KUKA KRL program: f1_Kuka_APT229T02S29.SRC

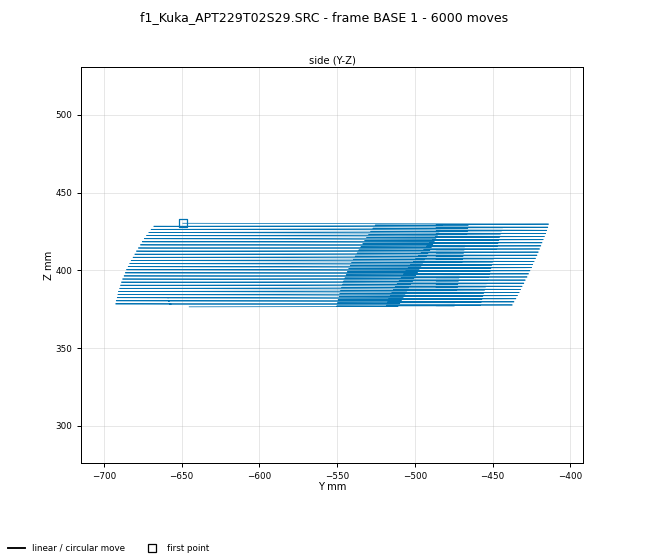
[picture p0: tool path of f1_Kuka_APT229T02S29.SRC in frame BASE 1, 6000 of 6001 moves have a stored position in this frame; points joined in program order, loops and branches not executed]
&ACCESS RVP
&REL 2
&PARAM TEMPLATE = C:\KRC\Roboter\Template\vorgabe
&PARAM EDITMASK = *
DEF f1_Kuka_APT229T02S29()


;FOLD INI;%{PE}%V3.2.0,%MKUKATPBASIS,%CINIT,%VCOMMON,%P
  ;FOLD BAS INI;%{E}%V3.2.0,%MKUKATPBASIS,%CINIT,%VINIT,%P
    GLOBAL INTERRUPT DECL 3 WHEN $STOPMESS==TRUE DO IR_STOPM ( )
    INTERRUPT ON 3
    BAS (#INITMOV,0 )
  ;ENDFOLD (BAS INI)
  ;FOLD USER INI;%{E}%V3.2.0,%MKUKATPUSER,%CINIT,%VINIT,%P
    ;Make your modifications here
  ;ENDFOLD (USER INI)
;ENDFOLD (INI)


;*** Make Null PTP Move
  PTP $pos_act

;*** Auto Load The Correct TOOL Data
  $tool=tool_data[2]

;*** Auto Load The Correct BASE Data
  $base=base_data[1]

  $ADVANCE = 5

;*** Restate Last Velocity
MMPM(30000.0)
SetRPM(8000)
LIN {X -0.016,Y -649.199,Z 430.291,A 0.000,B 0.000,C 90.000,E1 268.453} C_DIS
LIN {X 0.217,Y -646.027,Z 430.285,A 0.000,B 0.000,C 90.000,E1 267.192} C_DIS
LIN {X -0.248,Y -642.645,Z 430.278,A 0.000,B 0.000,C 90.000,E1 265.988} C_DIS
LIN {X 0.108,Y -637.908,Z 430.268,A 0.000,B 0.000,C 90.000,E1 264.204} C_DIS
LIN {X -0.169,Y -635.019,Z 430.262,A 0.000,B 0.000,C 90.000,E1 263.223} C_DIS
LIN {X -0.343,Y -630.490,Z 430.254,A 0.000,B 0.000,C 90.000,E1 261.724} C_DIS
LIN {X 0.198,Y -625.800,Z 430.245,A 0.000,B 0.000,C 90.000,E1 260.151} C_DIS
LIN {X 0.256,Y -621.879,Z 430.238,A 0.000,B 0.000,C 90.000,E1 258.870} C_DIS
LIN {X 0.011,Y -617.013,Z 430.230,A 0.000,B 0.000,C 90.000,E1 257.353} C_DIS
LIN {X 0.035,Y -612.805,Z 430.223,A 0.000,B 0.000,C 90.000,E1 256.061} C_DIS
LIN {X 0.137,Y -608.499,Z 430.215,A 0.000,B 0.000,C 90.000,E1 254.755} C_DIS
LIN {X 0.065,Y -603.102,Z 430.207,A 0.000,B 0.000,C 90.000,E1 253.196} C_DIS
LIN {X -0.110,Y -597.511,Z 430.198,A 0.000,B 0.000,C 90.000,E1 251.638} C_DIS
LIN {X -0.101,Y -592.747,Z 430.191,A 0.000,B 0.000,C 90.000,E1 250.315} C_DIS
LIN {X 0.225,Y -587.839,Z 430.183,A 0.000,B 0.000,C 90.000,E1 248.954} C_DIS
LIN {X -0.158,Y -583.761,Z 430.177,A 0.000,B 0.000,C 90.000,E1 247.922} C_DIS
LIN {X 0.241,Y -578.506,Z 430.170,A 0.000,B 0.000,C 90.000,E1 246.538} C_DIS
LIN {X -0.209,Y -573.098,Z 430.162,A 0.000,B 0.000,C 90.000,E1 245.229} C_DIS
LIN {X 0.076,Y -566.512,Z 430.153,A 0.000,B 0.000,C 90.000,E1 243.563} C_DIS
LIN {X -0.343,Y -561.046,Z 430.146,A 0.000,B 0.000,C 90.000,E1 242.231} C_DIS
LIN {X -0.009,Y -553.450,Z 430.135,A 0.000,B 0.000,C 90.000,E1 240.255} C_DIS
LIN {X 0.126,Y -546.096,Z 430.124,A 0.000,B 0.000,C 90.000,E1 238.280} C_DIS
LIN {X 0.161,Y -539.936,Z 430.114,A 0.000,B 0.000,C 90.000,E1 236.580} C_DIS
LIN {X -0.077,Y -532.802,Z 430.103,A 0.000,B 0.000,C 90.000,E1 234.609} C_DIS
LIN {X 0.300,Y -527.842,Z 430.095,A 0.000,B 0.000,C 90.000,E1 233.130} C_DIS
LIN {X 0.113,Y -521.840,Z 430.086,A 0.000,B 0.000,C 90.000,E1 231.412} C_DIS
LIN {X -0.126,Y -510.774,Z 430.066,A 0.000,B 0.000,C 90.000,E1 227.919} C_DIS
LIN {X -0.080,Y -505.592,Z 430.056,A 0.000,B 0.000,C 90.000,E1 226.134} C_DIS
LIN {X -0.164,Y -500.522,Z 430.046,A 0.000,B 0.000,C 90.000,E1 224.352} C_DIS
LIN {X 0.181,Y -494.664,Z 430.035,A 0.000,B 0.000,C 90.000,E1 222.204} C_DIS
LIN {X 0.227,Y -491.411,Z 430.028,A 0.000,B 0.000,C 90.000,E1 220.987} C_DIS
LIN {X 0.238,Y -485.107,Z 430.014,A 0.000,B 0.000,C 90.000,E1 218.543} C_DIS
LIN {X -0.168,Y -482.013,Z 430.008,A 0.000,B 0.000,C 90.000,E1 217.363} C_DIS
LIN {X -0.047,Y -478.278,Z 429.999,A 0.000,B 0.000,C 90.000,E1 215.804} C_DIS
LIN {X 0.000,Y -474.711,Z 429.990,A 0.000,B 0.000,C 90.000,E1 214.246} C_DIS
LIN {X 0.270,Y -470.560,Z 429.980,A 0.000,B 0.000,C 90.000,E1 212.339} C_DIS
LIN {X 0.198,Y -466.398,Z 429.969,A 0.000,B 0.000,C 90.000,E1 210.463} C_DIS
LIN {X 0.152,Y -463.698,Z 429.962,A 0.000,B 0.000,C 90.000,E1 209.205} C_DIS
LIN {X -0.031,Y -460.266,Z 429.954,A 0.000,B 0.000,C 90.000,E1 207.641} C_DIS
LIN {X -0.073,Y -455.343,Z 429.941,A 0.000,B 0.000,C 90.000,E1 205.412} C_DIS
LIN {X 0.200,Y -451.801,Z 429.932,A 0.000,B 0.000,C 90.000,E1 203.770} C_DIS
LIN {X 0.098,Y -447.565,Z 429.921,A 0.000,B 0.000,C 90.000,E1 201.844} C_DIS
LIN {X 0.136,Y -441.419,Z 429.905,A 0.000,B 0.000,C 90.000,E1 198.906} C_DIS
LIN {X -0.038,Y -436.063,Z 429.889,A 0.000,B 0.000,C 90.000,E1 195.969} C_DIS
LIN {X -0.014,Y -432.177,Z 429.876,A 0.000,B 0.000,C 90.000,E1 193.647} C_DIS
LIN {X -0.008,Y -427.119,Z 429.857,A 0.000,B 0.000,C 90.000,E1 190.310} C_DIS
LIN {X -0.166,Y -423.653,Z 429.842,A 0.000,B 0.000,C 90.000,E1 187.644} C_DIS
LIN {X -0.143,Y -420.857,Z 429.829,A 0.000,B 0.000,C 90.000,E1 185.277} C_DIS
LIN {X 0.063,Y -419.125,Z 429.820,A 0.000,B 0.000,C 90.000,E1 183.555} C_DIS
LIN {X -0.120,Y -416.780,Z 429.805,A 0.000,B 0.000,C 90.000,E1 180.859} C_DIS
LIN {X 0.009,Y -415.250,Z 429.791,A 0.000,B 0.000,C 90.000,E1 178.453} C_DIS
LIN {X 0.188,Y -414.001,Z 429.772,A 0.000,B 0.000,C 90.000,E1 175.008} C_DIS
LIN {X 0.130,Y -413.945,Z 429.750,A 0.000,B 0.000,C 90.000,E1 170.905} C_DIS
LIN {X 0.120,Y -414.832,Z 429.733,A 0.000,B 0.000,C 90.000,E1 167.825} C_DIS
LIN {X -0.129,Y -417.090,Z 429.712,A 0.000,B 0.000,C 90.000,E1 164.102} C_DIS
LIN {X -0.134,Y -419.840,Z 429.695,A 0.000,B 0.000,C 90.000,E1 161.040} C_DIS
LIN {X 0.203,Y -422.896,Z 429.680,A 0.000,B 0.000,C 90.000,E1 158.284} C_DIS
LIN {X 0.016,Y -426.446,Z 429.665,A 0.000,B 0.000,C 90.000,E1 155.613} C_DIS
LIN {X 0.098,Y -429.955,Z 429.652,A 0.000,B 0.000,C 90.000,E1 153.256} C_DIS
LIN {X -0.105,Y -432.179,Z 429.644,A 0.000,B 0.000,C 90.000,E1 151.948} C_DIS
LIN {X -0.048,Y -436.379,Z 429.631,A 0.000,B 0.000,C 90.000,E1 149.616} C_DIS
LIN {X 0.080,Y -441.687,Z 429.617,A 0.000,B 0.000,C 90.000,E1 146.962} C_DIS
LIN {X -0.047,Y -446.659,Z 429.604,A 0.000,B 0.000,C 90.000,E1 144.689} C_DIS
LIN {X -0.105,Y -454.457,Z 429.586,A 0.000,B 0.000,C 90.000,E1 141.457} C_DIS
LIN {X 0.086,Y -458.636,Z 429.577,A 0.000,B 0.000,C 90.000,E1 139.828} C_DIS
LIN {X 0.005,Y -462.850,Z 429.568,A 0.000,B 0.000,C 90.000,E1 138.243} C_DIS
LIN {X -0.151,Y -465.356,Z 429.563,A 0.000,B 0.000,C 90.000,E1 137.310} C_DIS
LIN {X -0.213,Y -468.530,Z 429.556,A 0.000,B 0.000,C 90.000,E1 136.053} C_DIS
LIN {X 0.190,Y -472.118,Z 429.547,A 0.000,B 0.000,C 90.000,E1 134.433} C_DIS
LIN {X -0.110,Y -474.684,Z 429.540,A 0.000,B 0.000,C 90.000,E1 133.218} C_DIS
LIN {X -0.237,Y -475.760,Z 429.537,A 0.000,B 0.000,C 90.000,E1 132.609} C_DIS
LIN {X -0.249,Y -477.194,Z 429.531,A 0.000,B 0.000,C 90.000,E1 131.676} C_DIS
LIN {X 0.115,Y -478.293,Z 429.526,A 0.000,B 0.000,C 90.000,E1 130.701} C_DIS
LIN {X -0.181,Y -478.951,Z 429.521,A 0.000,B 0.000,C 90.000,E1 129.806} C_DIS
LIN {X -0.074,Y -479.116,Z 429.519,A 0.000,B 0.000,C 90.000,E1 129.483} C_DIS
LIN {X 0.010,Y -479.158,Z 429.514,A 0.000,B 0.000,C 90.000,E1 128.543} C_DIS
LIN {X 0.097,Y -478.631,Z 429.509,A 0.000,B 0.000,C 90.000,E1 127.604} C_DIS
LIN {X 0.180,Y -477.585,Z 429.504,A 0.000,B 0.000,C 90.000,E1 126.664} C_DIS
LIN {X 0.246,Y -476.278,Z 429.499,A 0.000,B 0.000,C 90.000,E1 125.724} C_DIS
LIN {X 0.224,Y -475.231,Z 429.495,A 0.000,B 0.000,C 90.000,E1 125.105} C_DIS
LIN {X -0.193,Y -473.865,Z 429.492,A 0.000,B 0.000,C 90.000,E1 124.532} C_DIS
LIN {X -0.054,Y -471.563,Z 429.487,A 0.000,B 0.000,C 90.000,E1 123.579} C_DIS
LIN {X 0.061,Y -468.905,Z 429.481,A 0.000,B 0.000,C 90.000,E1 122.625} C_DIS
LIN {X -0.103,Y -464.908,Z 429.474,A 0.000,B 0.000,C 90.000,E1 121.386} C_DIS
LIN {X 0.090,Y -461.619,Z 429.469,A 0.000,B 0.000,C 90.000,E1 120.413} C_DIS
LIN {X -0.027,Y -456.831,Z 429.462,A 0.000,B 0.000,C 90.000,E1 119.155} C_DIS
LIN {X -0.090,Y -451.157,Z 429.454,A 0.000,B 0.000,C 90.000,E1 117.719} C_DIS
LIN {X 0.140,Y -445.297,Z 429.446,A 0.000,B 0.000,C 90.000,E1 116.232} C_DIS
LIN {X 0.209,Y -442.718,Z 429.442,A 0.000,B 0.000,C 90.000,E1 115.591} C_DIS
LIN {X 0.169,Y -442.732,Z 429.442,A 0.000,B 0.000,C 90.000,E1 115.591} C_DIS
LIN {X -0.059,Y -444.742,Z 429.439,A 0.000,B 0.000,C 90.000,E1 114.951} C_DIS
LIN {X -0.088,Y -454.712,Z 429.415,A 0.000,B 0.000,C 90.000,E1 110.737} C_DIS
LIN {X 0.035,Y -457.355,Z 429.410,A 0.000,B 0.000,C 90.000,E1 109.758} C_DIS
LIN {X 0.120,Y -465.984,Z 429.387,A 0.000,B 0.000,C 90.000,E1 105.607} C_DIS
LIN {X -0.158,Y -467.550,Z 429.383,A 0.000,B 0.000,C 90.000,E1 105.009} C_DIS
LIN {X 0.026,Y -468.567,Z 429.380,A 0.000,B 0.000,C 90.000,E1 104.356} C_DIS
LIN {X -0.215,Y -475.787,Z 429.357,A 0.000,B 0.000,C 90.000,E1 100.310} C_DIS
LIN {X 0.091,Y -476.298,Z 429.355,A 0.000,B 0.000,C 90.000,E1 99.962} C_DIS
LIN {X 0.039,Y -481.778,Z 429.331,A 0.000,B 0.000,C 90.000,E1 95.625} C_DIS
LIN {X -0.114,Y -482.169,Z 429.330,A 0.000,B 0.000,C 90.000,E1 95.334} C_DIS
LIN {X -0.185,Y -485.300,Z 429.306,A 0.000,B 0.000,C 90.000,E1 91.031} C_DIS
LIN {X 0.125,Y -485.537,Z 429.304,A 0.000,B 0.000,C 90.000,E1 90.688} C_DIS
LIN {X -0.153,Y -486.316,Z 429.282,A 0.000,B 0.000,C 90.000,E1 86.731} C_DIS
LIN {X -0.018,Y -486.309,Z 429.278,A 0.000,B 0.000,C 90.000,E1 86.102} C_DIS
LIN {X 0.186,Y -484.696,Z 429.255,A 0.000,B 0.000,C 90.000,E1 81.781} C_DIS
LIN {X 0.055,Y -484.608,Z 429.253,A 0.000,B 0.000,C 90.000,E1 81.489} C_DIS
LIN {X -0.065,Y -480.540,Z 429.227,A 0.000,B 0.000,C 90.000,E1 76.881} C_DIS
LIN {X -0.154,Y -474.292,Z 429.201,A 0.000,B 0.000,C 90.000,E1 72.236} C_DIS
LIN {X 0.117,Y -473.862,Z 429.200,A 0.000,B 0.000,C 90.000,E1 71.891} C_DIS
LIN {X -0.206,Y -466.265,Z 429.175,A 0.000,B 0.000,C 90.000,E1 67.539} C_DIS
LIN {X -0.277,Y -465.558,Z 429.172,A 0.000,B 0.000,C 90.000,E1 67.050} C_DIS
LIN {X 0.111,Y -465.576,Z 429.172,A 0.000,B 0.000,C 90.000,E1 66.997} C_DIS
LIN {X -0.066,Y -477.055,Z 429.164,A 0.000,B 0.000,C 90.000,E1 65.485} C_DIS
LIN {X -0.139,Y -485.128,Z 429.158,A 0.000,B 0.000,C 90.000,E1 64.409} C_DIS
LIN {X 0.101,Y -491.924,Z 429.153,A 0.000,B 0.000,C 90.000,E1 63.461} C_DIS
LIN {X -0.263,Y -497.100,Z 429.148,A 0.000,B 0.000,C 90.000,E1 62.743} C_DIS
LIN {X 0.056,Y -500.940,Z 429.145,A 0.000,B 0.000,C 90.000,E1 62.103} C_DIS
LIN {X -0.038,Y -504.550,Z 429.142,A 0.000,B 0.000,C 90.000,E1 61.513} C_DIS
LIN {X -0.104,Y -507.850,Z 429.138,A 0.000,B 0.000,C 90.000,E1 60.923} C_DIS
LIN {X -0.146,Y -510.859,Z 429.135,A 0.000,B 0.000,C 90.000,E1 60.333} C_DIS
LIN {X 0.010,Y -513.067,Z 429.133,A 0.000,B 0.000,C 90.000,E1 59.871} C_DIS
LIN {X 0.004,Y -515.608,Z 429.129,A 0.000,B 0.000,C 90.000,E1 59.282} C_DIS
LIN {X 0.281,Y -517.787,Z 429.126,A 0.000,B 0.000,C 90.000,E1 58.663} C_DIS
LIN {X -0.065,Y -518.781,Z 429.124,A 0.000,B 0.000,C 90.000,E1 58.408} C_DIS
LIN {X 0.238,Y -520.483,Z 429.121,A 0.000,B 0.000,C 90.000,E1 57.788} C_DIS
LIN {X 0.223,Y -522.504,Z 429.116,A 0.000,B 0.000,C 90.000,E1 56.914} C_DIS
LIN {X 0.124,Y -523.546,Z 429.113,A 0.000,B 0.000,C 90.000,E1 56.342} C_DIS
LIN {X 0.136,Y -524.629,Z 429.108,A 0.000,B 0.000,C 90.000,E1 55.468} C_DIS
LIN {X 0.023,Y -525.268,Z 429.103,A 0.000,B 0.000,C 90.000,E1 54.609} C_DIS
LIN {X -0.076,Y -525.472,Z 429.099,A 0.000,B 0.000,C 90.000,E1 53.749} C_DIS
LIN {X 0.248,Y -525.326,Z 429.094,A 0.000,B 0.000,C 90.000,E1 52.844} C_DIS
LIN {X 0.145,Y -524.993,Z 429.089,A 0.000,B 0.000,C 90.000,E1 51.984} C_DIS
LIN {X 0.326,Y -524.156,Z 429.082,A 0.000,B 0.000,C 90.000,E1 50.803} C_DIS
LIN {X 0.094,Y -523.105,Z 429.076,A 0.000,B 0.000,C 90.000,E1 49.666} C_DIS
LIN {X -0.149,Y -521.838,Z 429.070,A 0.000,B 0.000,C 90.000,E1 48.528} C_DIS
LIN {X 0.322,Y -520.387,Z 429.063,A 0.000,B 0.000,C 90.000,E1 47.310} C_DIS
LIN {X 0.219,Y -518.084,Z 429.053,A 0.000,B 0.000,C 90.000,E1 45.567} C_DIS
LIN {X -0.032,Y -515.626,Z 429.042,A 0.000,B 0.000,C 90.000,E1 43.542} C_DIS
LIN {X 0.137,Y -513.685,Z 429.032,A 0.000,B 0.000,C 90.000,E1 41.757} C_DIS
LIN {X -0.162,Y -511.433,Z 429.021,A 0.000,B 0.000,C 90.000,E1 39.725} C_DIS
LIN {X 0.050,Y -509.857,Z 429.012,A 0.000,B 0.000,C 90.000,E1 38.222} C_DIS
LIN {X -0.088,Y -507.810,Z 429.003,A 0.000,B 0.000,C 90.000,E1 36.457} C_DIS
LIN {X 0.132,Y -506.032,Z 428.994,A 0.000,B 0.000,C 90.000,E1 34.945} C_DIS
LIN {X -0.156,Y -504.549,Z 428.988,A 0.000,B 0.000,C 90.000,E1 33.785} C_DIS
LIN {X -0.272,Y -502.186,Z 428.978,A 0.000,B 0.000,C 90.000,E1 32.005} C_DIS
LIN {X -0.281,Y -499.794,Z 428.968,A 0.000,B 0.000,C 90.000,E1 30.207} C_DIS
LIN {X 0.199,Y -498.176,Z 428.961,A 0.000,B 0.000,C 90.000,E1 28.949} C_DIS
LIN {X -0.153,Y -495.846,Z 428.951,A 0.000,B 0.000,C 90.000,E1 27.180} C_DIS
LIN {X 0.137,Y -493.409,Z 428.939,A 0.000,B 0.000,C 90.000,E1 25.027} C_DIS
LIN {X -0.177,Y -490.454,Z 428.922,A 0.000,B 0.000,C 90.000,E1 22.025} C_DIS
LIN {X -0.133,Y -488.913,Z 428.910,A 0.000,B 0.000,C 90.000,E1 19.885} C_DIS
LIN {X -0.155,Y -487.703,Z 428.900,A 0.000,B 0.000,C 90.000,E1 18.055} C_DIS
LIN {X 0.085,Y -486.635,Z 428.892,A 0.000,B 0.000,C 90.000,E1 16.496} C_DIS
LIN {X 0.036,Y -485.106,Z 428.880,A 0.000,B 0.000,C 90.000,E1 14.356} C_DIS
LIN {X 0.027,Y -483.620,Z 428.864,A 0.000,B 0.000,C 90.000,E1 11.591} C_DIS
LIN {X -0.164,Y -483.028,Z 428.856,A 0.000,B 0.000,C 90.000,E1 10.074} C_DIS
LIN {X 0.025,Y -482.452,Z 428.842,A 0.000,B 0.000,C 90.000,E1 7.587} C_DIS
LIN {X -0.200,Y -482.436,Z 428.825,A 0.000,B 0.000,C 90.000,E1 4.531} C_DIS
LIN {X -0.119,Y -483.946,Z 428.803,A 0.000,B 0.000,C 90.000,E1 0.516} C_DIS
LIN {X 0.070,Y -488.037,Z 428.778,A 0.000,B 0.000,C 90.000,E1 356.102} C_DIS
LIN {X -0.152,Y -491.259,Z 428.765,A 0.000,B 0.000,C 90.000,E1 353.685} C_DIS
LIN {X -0.054,Y -494.482,Z 428.753,A 0.000,B 0.000,C 90.000,E1 351.546} C_DIS
LIN {X 0.208,Y -498.075,Z 428.741,A 0.000,B 0.000,C 90.000,E1 349.398} C_DIS
LIN {X -0.115,Y -507.281,Z 428.716,A 0.000,B 0.000,C 90.000,E1 344.936} C_DIS
LIN {X -0.011,Y -511.555,Z 428.706,A 0.000,B 0.000,C 90.000,E1 343.142} C_DIS
LIN {X -0.046,Y -517.550,Z 428.693,A 0.000,B 0.000,C 90.000,E1 340.786} C_DIS
LIN {X -0.153,Y -520.743,Z 428.687,A 0.000,B 0.000,C 90.000,E1 339.625} C_DIS
LIN {X 0.277,Y -526.392,Z 428.675,A 0.000,B 0.000,C 90.000,E1 337.539} C_DIS
LIN {X -0.110,Y -531.281,Z 428.666,A 0.000,B 0.000,C 90.000,E1 335.845} C_DIS
LIN {X 0.243,Y -537.947,Z 428.653,A 0.000,B 0.000,C 90.000,E1 333.512} C_DIS
LIN {X -0.164,Y -543.002,Z 428.644,A 0.000,B 0.000,C 90.000,E1 331.847} C_DIS
LIN {X 0.052,Y -548.210,Z 428.634,A 0.000,B 0.000,C 90.000,E1 330.127} C_DIS
LIN {X -0.132,Y -552.587,Z 428.626,A 0.000,B 0.000,C 90.000,E1 328.742} C_DIS
LIN {X 0.112,Y -557.674,Z 428.617,A 0.000,B 0.000,C 90.000,E1 327.041} C_DIS
LIN {X 0.102,Y -563.555,Z 428.606,A 0.000,B 0.000,C 90.000,E1 325.102} C_DIS
LIN {X -0.017,Y -568.641,Z 428.597,A 0.000,B 0.000,C 90.000,E1 323.463} C_DIS
LIN {X -0.030,Y -573.779,Z 428.588,A 0.000,B 0.000,C 90.000,E1 321.823} C_DIS
LIN {X -0.035,Y -579.108,Z 428.579,A 0.000,B 0.000,C 90.000,E1 320.194} C_DIS
LIN {X -0.105,Y -583.629,Z 428.571,A 0.000,B 0.000,C 90.000,E1 318.852} C_DIS
LIN {X 0.035,Y -588.923,Z 428.562,A 0.000,B 0.000,C 90.000,E1 317.229} C_DIS
LIN {X 0.087,Y -593.419,Z 428.555,A 0.000,B 0.000,C 90.000,E1 315.891} C_DIS
LIN {X -0.211,Y -597.918,Z 428.548,A 0.000,B 0.000,C 90.000,E1 314.595} C_DIS
LIN {X -0.003,Y -604.205,Z 428.537,A 0.000,B 0.000,C 90.000,E1 312.732} C_DIS
LIN {X -0.102,Y -608.674,Z 428.530,A 0.000,B 0.000,C 90.000,E1 311.434} C_DIS
LIN {X 0.344,Y -613.019,Z 428.523,A 0.000,B 0.000,C 90.000,E1 310.092} C_DIS
LIN {X 0.005,Y -617.270,Z 428.516,A 0.000,B 0.000,C 90.000,E1 308.830} C_DIS
LIN {X 0.051,Y -622.202,Z 428.507,A 0.000,B 0.000,C 90.000,E1 307.282} C_DIS
LIN {X 0.134,Y -625.268,Z 428.502,A 0.000,B 0.000,C 90.000,E1 306.251} C_DIS
LIN {X -0.048,Y -629.805,Z 428.493,A 0.000,B 0.000,C 90.000,E1 304.739} C_DIS
LIN {X 0.166,Y -633.388,Z 428.486,A 0.000,B 0.000,C 90.000,E1 303.452} C_DIS
LIN {X -0.083,Y -636.910,Z 428.479,A 0.000,B 0.000,C 90.000,E1 302.212} C_DIS
LIN {X 0.256,Y -640.311,Z 428.472,A 0.000,B 0.000,C 90.000,E1 300.924} C_DIS
LIN {X -0.171,Y -644.131,Z 428.464,A 0.000,B 0.000,C 90.000,E1 299.461} C_DIS
LIN {X -0.358,Y -647.179,Z 428.457,A 0.000,B 0.000,C 90.000,E1 298.231} C_DIS
LIN {X 0.183,Y -650.635,Z 428.448,A 0.000,B 0.000,C 90.000,E1 296.693} C_DIS
LIN {X 0.102,Y -653.383,Z 428.442,A 0.000,B 0.000,C 90.000,E1 295.463} C_DIS
LIN {X -0.228,Y -655.906,Z 428.435,A 0.000,B 0.000,C 90.000,E1 294.259} C_DIS
LIN {X -0.181,Y -658.221,Z 428.428,A 0.000,B 0.000,C 90.000,E1 293.025} C_DIS
LIN {X 0.161,Y -660.404,Z 428.421,A 0.000,B 0.000,C 90.000,E1 291.770} C_DIS
LIN {X 0.161,Y -662.106,Z 428.416,A 0.000,B 0.000,C 90.000,E1 290.791} C_DIS
LIN {X 0.185,Y -663.600,Z 428.410,A 0.000,B 0.000,C 90.000,E1 289.812} C_DIS
LIN {X 0.126,Y -665.027,Z 428.403,A 0.000,B 0.000,C 90.000,E1 288.598} C_DIS
LIN {X -0.004,Y -666.380,Z 428.395,A 0.000,B 0.000,C 90.000,E1 287.149} C_DIS
LIN {X -0.334,Y -666.984,Z 428.390,A 0.000,B 0.000,C 90.000,E1 286.205} C_DIS
LIN {X 0.176,Y -667.471,Z 428.385,A 0.000,B 0.000,C 90.000,E1 285.190} C_DIS
LIN {X -0.201,Y -667.826,Z 428.378,A 0.000,B 0.000,C 90.000,E1 284.008} C_DIS
LIN {X 0.077,Y -667.853,Z 428.371,A 0.000,B 0.000,C 90.000,E1 282.771} C_DIS
LIN {X -0.227,Y -667.796,Z 428.366,A 0.000,B 0.000,C 90.000,E1 281.827} C_DIS
LIN {X -0.017,Y -667.526,Z 428.360,A 0.000,B 0.000,C 90.000,E1 280.838} C_DIS
LIN {X 0.195,Y -667.169,Z 428.355,A 0.000,B 0.000,C 90.000,E1 279.849} C_DIS
LIN {X -0.258,Y -666.520,Z 428.349,A 0.000,B 0.000,C 90.000,E1 278.916} C_DIS
LIN {X 0.302,Y -665.478,Z 428.341,A 0.000,B 0.000,C 90.000,E1 277.409} C_DIS
LIN {X -0.277,Y -664.604,Z 428.336,A 0.000,B 0.000,C 90.000,E1 276.486} C_DIS
LIN {X 0.087,Y -662.846,Z 428.328,A 0.000,B 0.000,C 90.000,E1 274.992} C_DIS
LIN {X 0.127,Y -661.526,Z 428.322,A 0.000,B 0.000,C 90.000,E1 274.012} C_DIS
LIN {X -0.236,Y -660.847,Z 428.320,A 0.000,B 0.000,C 90.000,E1 273.555} C_DIS
LIN {X -0.166,Y -657.885,Z 428.310,A 0.000,B 0.000,C 90.000,E1 271.835} C_DIS
LIN {X 0.221,Y -655.564,Z 428.303,A 0.000,B 0.000,C 90.000,E1 270.573} C_DIS
LIN {X -0.102,Y -652.947,Z 428.297,A 0.000,B 0.000,C 90.000,E1 269.370} C_DIS
LIN {X -0.264,Y -650.618,Z 428.291,A 0.000,B 0.000,C 90.000,E1 268.396} C_DIS
LIN {X -0.006,Y -647.462,Z 428.284,A 0.000,B 0.000,C 90.000,E1 267.135} C_DIS
LIN {X 0.007,Y -643.381,Z 428.276,A 0.000,B 0.000,C 90.000,E1 265.641} C_DIS
LIN {X 0.192,Y -640.075,Z 428.269,A 0.000,B 0.000,C 90.000,E1 264.375} C_DIS
LIN {X -0.317,Y -636.524,Z 428.262,A 0.000,B 0.000,C 90.000,E1 263.166} C_DIS
LIN {X 0.254,Y -631.946,Z 428.254,A 0.000,B 0.000,C 90.000,E1 261.602} C_DIS
LIN {X -0.309,Y -628.021,Z 428.246,A 0.000,B 0.000,C 90.000,E1 260.387} C_DIS
LIN {X -0.215,Y -624.113,Z 428.239,A 0.000,B 0.000,C 90.000,E1 259.106} C_DIS
LIN {X 0.323,Y -619.233,Z 428.231,A 0.000,B 0.000,C 90.000,E1 257.521} C_DIS
LIN {X 0.027,Y -615.929,Z 428.225,A 0.000,B 0.000,C 90.000,E1 256.520} C_DIS
LIN {X -0.208,Y -610.780,Z 428.217,A 0.000,B 0.000,C 90.000,E1 254.991} C_DIS
LIN {X 0.352,Y -605.388,Z 428.208,A 0.000,B 0.000,C 90.000,E1 253.378} C_DIS
LIN {X -0.253,Y -600.766,Z 428.201,A 0.000,B 0.000,C 90.000,E1 252.127} C_DIS
LIN {X 0.006,Y -596.023,Z 428.193,A 0.000,B 0.000,C 90.000,E1 250.786} C_DIS
LIN {X 0.189,Y -591.135,Z 428.186,A 0.000,B 0.000,C 90.000,E1 249.444} C_DIS
LIN {X -0.265,Y -586.084,Z 428.179,A 0.000,B 0.000,C 90.000,E1 248.156} C_DIS
LIN {X -0.046,Y -580.839,Z 428.171,A 0.000,B 0.000,C 90.000,E1 246.794} C_DIS
LIN {X 0.067,Y -575.416,Z 428.164,A 0.000,B 0.000,C 90.000,E1 245.433} C_DIS
LIN {X -0.122,Y -568.821,Z 428.155,A 0.000,B 0.000,C 90.000,E1 243.819} C_DIS
LIN {X 0.262,Y -563.346,Z 428.147,A 0.000,B 0.000,C 90.000,E1 242.410} C_DIS
LIN {X 0.165,Y -554.657,Z 428.135,A 0.000,B 0.000,C 90.000,E1 240.205} C_DIS
LIN {X 0.140,Y -547.264,Z 428.124,A 0.000,B 0.000,C 90.000,E1 238.250} C_DIS
LIN {X -0.084,Y -541.117,Z 428.114,A 0.000,B 0.000,C 90.000,E1 236.580} C_DIS
LIN {X 0.144,Y -533.045,Z 428.102,A 0.000,B 0.000,C 90.000,E1 234.276} C_DIS
LIN {X 0.095,Y -528.088,Z 428.094,A 0.000,B 0.000,C 90.000,E1 232.844} C_DIS
LIN {X -0.045,Y -523.100,Z 428.086,A 0.000,B 0.000,C 90.000,E1 231.412} C_DIS
LIN {X 0.152,Y -511.992,Z 428.066,A 0.000,B 0.000,C 90.000,E1 227.877} C_DIS
LIN {X 0.081,Y -505.962,Z 428.055,A 0.000,B 0.000,C 90.000,E1 225.810} C_DIS
LIN {X 0.215,Y -500.042,Z 428.043,A 0.000,B 0.000,C 90.000,E1 223.704} C_DIS
LIN {X 0.204,Y -494.262,Z 428.031,A 0.000,B 0.000,C 90.000,E1 221.595} C_DIS
LIN {X -0.078,Y -487.834,Z 428.018,A 0.000,B 0.000,C 90.000,E1 219.197} C_DIS
LIN {X 0.064,Y -483.985,Z 428.009,A 0.000,B 0.000,C 90.000,E1 217.649} C_DIS
LIN {X 0.031,Y -479.463,Z 427.999,A 0.000,B 0.000,C 90.000,E1 215.804} C_DIS
LIN {X 0.287,Y -475.161,Z 427.989,A 0.000,B 0.000,C 90.000,E1 213.913} C_DIS
LIN {X -0.254,Y -471.705,Z 427.980,A 0.000,B 0.000,C 90.000,E1 212.418} C_DIS
LIN {X -0.133,Y -466.844,Z 427.968,A 0.000,B 0.000,C 90.000,E1 210.207} C_DIS
LIN {X -0.026,Y -463.423,Z 427.959,A 0.000,B 0.000,C 90.000,E1 208.615} C_DIS
LIN {X 0.070,Y -460.642,Z 427.952,A 0.000,B 0.000,C 90.000,E1 207.334} C_DIS
LIN {X 0.141,Y -456.396,Z 427.941,A 0.000,B 0.000,C 90.000,E1 205.412} C_DIS
LIN {X 0.019,Y -452.833,Z 427.932,A 0.000,B 0.000,C 90.000,E1 203.823} C_DIS
LIN {X 0.053,Y -449.257,Z 427.923,A 0.000,B 0.000,C 90.000,E1 202.206} C_DIS
LIN {X 0.005,Y -444.334,Z 427.911,A 0.000,B 0.000,C 90.000,E1 199.939} C_DIS
LIN {X -0.102,Y -438.086,Z 427.893,A 0.000,B 0.000,C 90.000,E1 196.677} C_DIS
LIN {X 0.166,Y -434.680,Z 427.882,A 0.000,B 0.000,C 90.000,E1 194.662} C_DIS
LIN {X 0.040,Y -430.907,Z 427.869,A 0.000,B 0.000,C 90.000,E1 192.355} C_DIS
LIN {X -0.064,Y -427.941,Z 427.858,A 0.000,B 0.000,C 90.000,E1 190.366} C_DIS
LIN {X 0.131,Y -424.855,Z 427.845,A 0.000,B 0.000,C 90.000,E1 187.992} C_DIS
LIN {X -0.157,Y -421.648,Z 427.830,A 0.000,B 0.000,C 90.000,E1 185.334} C_DIS
LIN {X 0.203,Y -418.647,Z 427.813,A 0.000,B 0.000,C 90.000,E1 182.236} C_DIS
LIN {X 0.036,Y -416.202,Z 427.794,A 0.000,B 0.000,C 90.000,E1 178.854} C_DIS
LIN {X -0.150,Y -414.691,Z 427.773,A 0.000,B 0.000,C 90.000,E1 175.122} C_DIS
LIN {X 0.058,Y -414.429,Z 427.758,A 0.000,B 0.000,C 90.000,E1 172.356} C_DIS
LIN {X 0.177,Y -414.624,Z 427.750,A 0.000,B 0.000,C 90.000,E1 170.971} C_DIS
LIN {X -0.144,Y -415.494,Z 427.733,A 0.000,B 0.000,C 90.000,E1 167.937} C_DIS
LIN {X 0.049,Y -417.772,Z 427.712,A 0.000,B 0.000,C 90.000,E1 164.157} C_DIS
LIN {X 0.076,Y -420.517,Z 427.695,A 0.000,B 0.000,C 90.000,E1 161.094} C_DIS
LIN {X 0.073,Y -423.969,Z 427.678,A 0.000,B 0.000,C 90.000,E1 158.050} C_DIS
LIN {X -0.103,Y -427.098,Z 427.665,A 0.000,B 0.000,C 90.000,E1 155.717} C_DIS
LIN {X -0.181,Y -430.654,Z 427.652,A 0.000,B 0.000,C 90.000,E1 153.384} C_DIS
LIN {X -0.127,Y -435.864,Z 427.635,A 0.000,B 0.000,C 90.000,E1 150.383} C_DIS
LIN {X 0.180,Y -441.780,Z 427.619,A 0.000,B 0.000,C 90.000,E1 147.375} C_DIS
LIN {X 0.058,Y -445.280,Z 427.610,A 0.000,B 0.000,C 90.000,E1 145.754} C_DIS
LIN {X -0.159,Y -449.760,Z 427.599,A 0.000,B 0.000,C 90.000,E1 143.829} C_DIS
LIN {X 0.178,Y -457.120,Z 427.583,A 0.000,B 0.000,C 90.000,E1 140.884} C_DIS
LIN {X 0.070,Y -461.412,Z 427.574,A 0.000,B 0.000,C 90.000,E1 139.299} C_DIS
LIN {X 0.041,Y -465.716,Z 427.565,A 0.000,B 0.000,C 90.000,E1 137.715} C_DIS
LIN {X 0.059,Y -469.788,Z 427.556,A 0.000,B 0.000,C 90.000,E1 136.134} C_DIS
LIN {X 0.061,Y -472.783,Z 427.549,A 0.000,B 0.000,C 90.000,E1 134.879} C_DIS
LIN {X 0.011,Y -474.819,Z 427.544,A 0.000,B 0.000,C 90.000,E1 133.947} C_DIS
LIN {X -0.011,Y -476.752,Z 427.539,A 0.000,B 0.000,C 90.000,E1 133.014} C_DIS
LIN {X 0.103,Y -478.776,Z 427.532,A 0.000,B 0.000,C 90.000,E1 131.757} C_DIS
LIN {X 0.011,Y -479.592,Z 427.529,A 0.000,B 0.000,C 90.000,E1 131.148} C_DIS
LIN {X -0.075,Y -480.298,Z 427.525,A 0.000,B 0.000,C 90.000,E1 130.539} C_DIS
LIN {X 0.020,Y -480.916,Z 427.520,A 0.000,B 0.000,C 90.000,E1 129.600} C_DIS
LIN {X 0.135,Y -481.095,Z 427.518,A 0.000,B 0.000,C 90.000,E1 129.277} C_DIS
LIN {X -0.133,Y -481.050,Z 427.513,A 0.000,B 0.000,C 90.000,E1 128.382} C_DIS
LIN {X -0.026,Y -480.436,Z 427.508,A 0.000,B 0.000,C 90.000,E1 127.443} C_DIS
LIN {X 0.074,Y -479.335,Z 427.503,A 0.000,B 0.000,C 90.000,E1 126.503} C_DIS
LIN {X -0.122,Y -478.003,Z 427.498,A 0.000,B 0.000,C 90.000,E1 125.598} C_DIS
LIN {X 0.146,Y -476.938,Z 427.494,A 0.000,B 0.000,C 90.000,E1 124.945} C_DIS
LIN {X -0.076,Y -474.750,Z 427.489,A 0.000,B 0.000,C 90.000,E1 124.040} C_DIS
LIN {X -0.107,Y -473.181,Z 427.486,A 0.000,B 0.000,C 90.000,E1 123.420} C_DIS
LIN {X 0.022,Y -470.439,Z 427.480,A 0.000,B 0.000,C 90.000,E1 122.467} C_DIS
LIN {X -0.128,Y -467.404,Z 427.475,A 0.000,B 0.000,C 90.000,E1 121.544} C_DIS
LIN {X -0.064,Y -464.182,Z 427.470,A 0.000,B 0.000,C 90.000,E1 120.590} C_DIS
LIN {X 0.102,Y -459.982,Z 427.464,A 0.000,B 0.000,C 90.000,E1 119.461} C_DIS
LIN {X 0.084,Y -454.305,Z 427.456,A 0.000,B 0.000,C 90.000,E1 118.025} C_DIS
LIN {X -0.115,Y -449.738,Z 427.450,A 0.000,B 0.000,C 90.000,E1 116.924} C_DIS
LIN {X -0.114,Y -443.700,Z 427.441,A 0.000,B 0.000,C 90.000,E1 115.463} C_DIS
LIN {X -0.227,Y -443.420,Z 427.441,A 0.000,B 0.000,C 90.000,E1 115.412} C_DIS
LIN {X -0.076,Y -443.434,Z 427.441,A 0.000,B 0.000,C 90.000,E1 115.387} C_DIS
LIN {X 0.189,Y -445.077,Z 427.438,A 0.000,B 0.000,C 90.000,E1 114.771} C_DIS
LIN {X -0.127,Y -454.237,Z 427.416,A 0.000,B 0.000,C 90.000,E1 110.918} C_DIS
LIN {X -0.011,Y -456.901,Z 427.411,A 0.000,B 0.000,C 90.000,E1 109.939} C_DIS
LIN {X -0.109,Y -457.615,Z 427.409,A 0.000,B 0.000,C 90.000,E1 109.631} C_DIS
LIN {X -0.023,Y -466.333,Z 427.386,A 0.000,B 0.000,C 90.000,E1 105.481} C_DIS
LIN {X 0.151,Y -467.870,Z 427.383,A 0.000,B 0.000,C 90.000,E1 104.828} C_DIS
LIN {X 0.179,Y -475.431,Z 427.358,A 0.000,B 0.000,C 90.000,E1 100.433} C_DIS
LIN {X 0.018,Y -476.081,Z 427.356,A 0.000,B 0.000,C 90.000,E1 100.141} C_DIS
LIN {X -0.179,Y -482.004,Z 427.331,A 0.000,B 0.000,C 90.000,E1 95.511} C_DIS
LIN {X -0.198,Y -482.514,Z 427.325,A 0.000,B 0.000,C 90.000,E1 94.588} C_DIS
LIN {X 0.092,Y -485.449,Z 427.305,A 0.000,B 0.000,C 90.000,E1 90.859} C_DIS
LIN {X 0.229,Y -485.505,Z 427.301,A 0.000,B 0.000,C 90.000,E1 90.229} C_DIS
LIN {X 0.125,Y -486.381,Z 427.281,A 0.000,B 0.000,C 90.000,E1 86.560} C_DIS
LIN {X -0.051,Y -486.365,Z 427.279,A 0.000,B 0.000,C 90.000,E1 86.274} C_DIS
LIN {X 0.038,Y -484.690,Z 427.254,A 0.000,B 0.000,C 90.000,E1 81.659} C_DIS
LIN {X 0.184,Y -484.073,Z 427.250,A 0.000,B 0.000,C 90.000,E1 81.027} C_DIS
LIN {X -0.161,Y -480.640,Z 427.228,A 0.000,B 0.000,C 90.000,E1 77.061} C_DIS
LIN {X -0.194,Y -480.346,Z 427.226,A 0.000,B 0.000,C 90.000,E1 76.756} C_DIS
LIN {X 0.177,Y -474.152,Z 427.200,A 0.000,B 0.000,C 90.000,E1 72.054} C_DIS
LIN {X 0.098,Y -465.895,Z 427.174,A 0.000,B 0.000,C 90.000,E1 67.230} C_DIS
LIN {X 0.058,Y -465.932,Z 427.174,A 0.000,B 0.000,C 90.000,E1 67.230} C_DIS
LIN {X 0.050,Y -479.069,Z 427.164,A 0.000,B 0.000,C 90.000,E1 65.485} C_DIS
LIN {X -0.210,Y -488.244,Z 427.157,A 0.000,B 0.000,C 90.000,E1 64.280} C_DIS
LIN {X -0.168,Y -493.847,Z 427.153,A 0.000,B 0.000,C 90.000,E1 63.512} C_DIS
LIN {X 0.127,Y -498.008,Z 427.149,A 0.000,B 0.000,C 90.000,E1 62.871} C_DIS
LIN {X 0.013,Y -501.879,Z 427.146,A 0.000,B 0.000,C 90.000,E1 62.281} C_DIS
LIN {X -0.071,Y -505.482,Z 427.143,A 0.000,B 0.000,C 90.000,E1 61.691} C_DIS
LIN {X -0.128,Y -508.812,Z 427.139,A 0.000,B 0.000,C 90.000,E1 61.101} C_DIS
LIN {X 0.284,Y -511.884,Z 427.136,A 0.000,B 0.000,C 90.000,E1 60.461} C_DIS
LIN {X -0.171,Y -514.738,Z 427.133,A 0.000,B 0.000,C 90.000,E1 59.921} C_DIS
LIN {X 0.108,Y -517.808,Z 427.129,A 0.000,B 0.000,C 90.000,E1 59.154} C_DIS
LIN {X -0.044,Y -519.912,Z 427.125,A 0.000,B 0.000,C 90.000,E1 58.584} C_DIS
LIN {X -0.004,Y -521.638,Z 427.122,A 0.000,B 0.000,C 90.000,E1 57.995} C_DIS
LIN {X -0.008,Y -523.742,Z 427.117,A 0.000,B 0.000,C 90.000,E1 57.120} C_DIS
LIN {X -0.099,Y -524.805,Z 427.114,A 0.000,B 0.000,C 90.000,E1 56.548} C_DIS
LIN {X -0.073,Y -525.937,Z 427.109,A 0.000,B 0.000,C 90.000,E1 55.674} C_DIS
LIN {X -0.172,Y -526.678,Z 427.104,A 0.000,B 0.000,C 90.000,E1 54.815} C_DIS
LIN {X 0.169,Y -526.900,Z 427.100,A 0.000,B 0.000,C 90.000,E1 53.909} C_DIS
LIN {X 0.086,Y -526.754,Z 427.095,A 0.000,B 0.000,C 90.000,E1 53.050} C_DIS
LIN {X 0.002,Y -526.426,Z 427.090,A 0.000,B 0.000,C 90.000,E1 52.190} C_DIS
LIN {X 0.206,Y -525.611,Z 427.084,A 0.000,B 0.000,C 90.000,E1 51.009} C_DIS
LIN {X 0.061,Y -524.555,Z 427.077,A 0.000,B 0.000,C 90.000,E1 49.865} C_DIS
LIN {X 0.127,Y -522.960,Z 427.069,A 0.000,B 0.000,C 90.000,E1 48.405} C_DIS
LIN {X -0.217,Y -521.049,Z 427.061,A 0.000,B 0.000,C 90.000,E1 46.986} C_DIS
LIN {X 0.266,Y -517.990,Z 427.048,A 0.000,B 0.000,C 90.000,E1 44.595} C_DIS
LIN {X 0.034,Y -515.592,Z 427.037,A 0.000,B 0.000,C 90.000,E1 42.567} C_DIS
LIN {X 0.289,Y -513.944,Z 427.028,A 0.000,B 0.000,C 90.000,E1 41.067} C_DIS
LIN {X 0.074,Y -512.034,Z 427.019,A 0.000,B 0.000,C 90.000,E1 39.322} C_DIS
LIN {X -0.028,Y -510.417,Z 427.010,A 0.000,B 0.000,C 90.000,E1 37.855} C_DIS
LIN {X -0.063,Y -508.684,Z 427.002,A 0.000,B 0.000,C 90.000,E1 36.377} C_DIS
LIN {X -0.119,Y -506.893,Z 426.994,A 0.000,B 0.000,C 90.000,E1 34.898} C_DIS
LIN {X -0.108,Y -505.394,Z 426.987,A 0.000,B 0.000,C 90.000,E1 33.706} C_DIS
LIN {X 0.215,Y -503.034,Z 426.977,A 0.000,B 0.000,C 90.000,E1 31.878} C_DIS
LIN {X -0.072,Y -501.030,Z 426.969,A 0.000,B 0.000,C 90.000,E1 30.413} C_DIS
LIN {X -0.108,Y -498.611,Z 426.959,A 0.000,B 0.000,C 90.000,E1 28.615} C_DIS
LIN {X 0.081,Y -495.643,Z 426.946,A 0.000,B 0.000,C 90.000,E1 26.181} C_DIS
LIN {X -0.028,Y -493.006,Z 426.932,A 0.000,B 0.000,C 90.000,E1 23.770} C_DIS
LIN {X -0.088,Y -490.416,Z 426.915,A 0.000,B 0.000,C 90.000,E1 20.737} C_DIS
LIN {X -0.048,Y -488.983,Z 426.903,A 0.000,B 0.000,C 90.000,E1 18.598} C_DIS
LIN {X 0.218,Y -487.921,Z 426.895,A 0.000,B 0.000,C 90.000,E1 17.040} C_DIS
LIN {X -0.135,Y -486.621,Z 426.885,A 0.000,B 0.000,C 90.000,E1 15.245} C_DIS
LIN {X -0.085,Y -484.929,Z 426.869,A 0.000,B 0.000,C 90.000,E1 12.479} C_DIS
LIN {X 0.068,Y -484.079,Z 426.857,A 0.000,B 0.000,C 90.000,E1 10.310} C_DIS
LIN {X 0.157,Y -483.407,Z 426.842,A 0.000,B 0.000,C 90.000,E1 7.530} C_DIS
LIN {X -0.215,Y -483.455,Z 426.823,A 0.000,B 0.000,C 90.000,E1 4.188} C_DIS
LIN {X -0.072,Y -485.157,Z 426.801,A 0.000,B 0.000,C 90.000,E1 0.172} C_DIS
LIN {X -0.016,Y -489.462,Z 426.777,A 0.000,B 0.000,C 90.000,E1 355.812} C_DIS
LIN {X -0.184,Y -492.744,Z 426.763,A 0.000,B 0.000,C 90.000,E1 353.394} C_DIS
LIN {X -0.038,Y -496.063,Z 426.751,A 0.000,B 0.000,C 90.000,E1 351.254} C_DIS
LIN {X -0.224,Y -499.711,Z 426.740,A 0.000,B 0.000,C 90.000,E1 349.162} C_DIS
LIN {X 0.169,Y -509.155,Z 426.715,A 0.000,B 0.000,C 90.000,E1 344.629} C_DIS
LIN {X 0.176,Y -513.411,Z 426.705,A 0.000,B 0.000,C 90.000,E1 342.851} C_DIS
LIN {X 0.087,Y -517.939,Z 426.695,A 0.000,B 0.000,C 90.000,E1 341.094} C_DIS
LIN {X -0.049,Y -521.891,Z 426.687,A 0.000,B 0.000,C 90.000,E1 339.645} C_DIS
LIN {X -0.065,Y -526.742,Z 426.677,A 0.000,B 0.000,C 90.000,E1 337.901} C_DIS
LIN {X -0.278,Y -533.244,Z 426.664,A 0.000,B 0.000,C 90.000,E1 335.613} C_DIS
LIN {X -0.096,Y -539.117,Z 426.653,A 0.000,B 0.000,C 90.000,E1 333.589} C_DIS
LIN {X -0.009,Y -545.067,Z 426.642,A 0.000,B 0.000,C 90.000,E1 331.591} C_DIS
LIN {X -0.253,Y -549.444,Z 426.634,A 0.000,B 0.000,C 90.000,E1 330.205} C_DIS
LIN {X -0.136,Y -553.872,Z 426.627,A 0.000,B 0.000,C 90.000,E1 328.791} C_DIS
LIN {X -0.078,Y -559.825,Z 426.616,A 0.000,B 0.000,C 90.000,E1 326.834} C_DIS
LIN {X -0.038,Y -565.750,Z 426.605,A 0.000,B 0.000,C 90.000,E1 324.895} C_DIS
LIN {X 0.217,Y -570.001,Z 426.597,A 0.000,B 0.000,C 90.000,E1 323.497} C_DIS
LIN {X -0.083,Y -576.056,Z 426.587,A 0.000,B 0.000,C 90.000,E1 321.618} C_DIS
LIN {X -0.209,Y -580.511,Z 426.579,A 0.000,B 0.000,C 90.000,E1 320.275} C_DIS
LIN {X -0.082,Y -585.941,Z 426.570,A 0.000,B 0.000,C 90.000,E1 318.647} C_DIS
LIN {X -0.145,Y -592.159,Z 426.560,A 0.000,B 0.000,C 90.000,E1 316.782} C_DIS
LIN {X -0.244,Y -595.772,Z 426.554,A 0.000,B 0.000,C 90.000,E1 315.729} C_DIS
LIN {X 0.345,Y -600.336,Z 426.547,A 0.000,B 0.000,C 90.000,E1 314.352} C_DIS
LIN {X -0.043,Y -605.732,Z 426.538,A 0.000,B 0.000,C 90.000,E1 312.813} C_DIS
LIN {X -0.115,Y -610.223,Z 426.531,A 0.000,B 0.000,C 90.000,E1 311.515} C_DIS
LIN {X -0.110,Y -614.606,Z 426.523,A 0.000,B 0.000,C 90.000,E1 310.216} C_DIS
LIN {X -0.120,Y -619.733,Z 426.515,A 0.000,B 0.000,C 90.000,E1 308.669} C_DIS
LIN {X 0.132,Y -623.870,Z 426.508,A 0.000,B 0.000,C 90.000,E1 307.363} C_DIS
LIN {X 0.081,Y -627.691,Z 426.501,A 0.000,B 0.000,C 90.000,E1 306.091} C_DIS
LIN {X 0.097,Y -631.494,Z 426.494,A 0.000,B 0.000,C 90.000,E1 304.818} C_DIS
LIN {X -0.185,Y -635.104,Z 426.487,A 0.000,B 0.000,C 90.000,E1 303.579} C_DIS
LIN {X 0.129,Y -638.675,Z 426.480,A 0.000,B 0.000,C 90.000,E1 302.291} C_DIS
LIN {X 0.012,Y -642.750,Z 426.471,A 0.000,B 0.000,C 90.000,E1 300.797} C_DIS
LIN {X 0.197,Y -646.609,Z 426.463,A 0.000,B 0.000,C 90.000,E1 299.283} C_DIS
LIN {X -0.031,Y -649.019,Z 426.457,A 0.000,B 0.000,C 90.000,E1 298.309} C_DIS
LIN {X -0.026,Y -652.498,Z 426.449,A 0.000,B 0.000,C 90.000,E1 296.821} C_DIS
LIN {X 0.036,Y -655.786,Z 426.441,A 0.000,B 0.000,C 90.000,E1 295.335} C_DIS
LIN {X 0.344,Y -658.315,Z 426.434,A 0.000,B 0.000,C 90.000,E1 294.079} C_DIS
LIN {X -0.047,Y -661.117,Z 426.426,A 0.000,B 0.000,C 90.000,E1 292.642} C_DIS
LIN {X 0.109,Y -664.025,Z 426.416,A 0.000,B 0.000,C 90.000,E1 290.918} C_DIS
LIN {X 0.160,Y -665.492,Z 426.411,A 0.000,B 0.000,C 90.000,E1 289.939} C_DIS
LIN {X 0.137,Y -666.922,Z 426.404,A 0.000,B 0.000,C 90.000,E1 288.725} C_DIS
LIN {X 0.130,Y -668.067,Z 426.397,A 0.000,B 0.000,C 90.000,E1 287.511} C_DIS
LIN {X -0.142,Y -668.926,Z 426.389,A 0.000,B 0.000,C 90.000,E1 286.079} C_DIS
LIN {X 0.216,Y -669.327,Z 426.384,A 0.000,B 0.000,C 90.000,E1 285.079} C_DIS
LIN {X 0.106,Y -669.603,Z 426.379,A 0.000,B 0.000,C 90.000,E1 284.120} C_DIS
LIN {X -0.245,Y -669.586,Z 426.372,A 0.000,B 0.000,C 90.000,E1 282.939} C_DIS
LIN {X -0.090,Y -669.396,Z 426.365,A 0.000,B 0.000,C 90.000,E1 281.715} C_DIS
LIN {X 0.072,Y -668.931,Z 426.358,A 0.000,B 0.000,C 90.000,E1 280.489} C_DIS
LIN {X -0.163,Y -668.593,Z 426.354,A 0.000,B 0.000,C 90.000,E1 279.782} C_DIS
LIN {X -0.136,Y -667.680,Z 426.348,A 0.000,B 0.000,C 90.000,E1 278.568} C_DIS
LIN {X -0.120,Y -666.750,Z 426.341,A 0.000,B 0.000,C 90.000,E1 277.352} C_DIS
LIN {X -0.020,Y -665.819,Z 426.335,A 0.000,B 0.000,C 90.000,E1 276.372} C_DIS
LIN {X -0.290,Y -664.107,Z 426.327,A 0.000,B 0.000,C 90.000,E1 274.935} C_DIS
LIN {X -0.232,Y -662.793,Z 426.322,A 0.000,B 0.000,C 90.000,E1 273.955} C_DIS
LIN {X 0.074,Y -662.105,Z 426.319,A 0.000,B 0.000,C 90.000,E1 273.440} C_DIS
LIN {X -0.304,Y -659.673,Z 426.311,A 0.000,B 0.000,C 90.000,E1 272.007} C_DIS
LIN {X -0.074,Y -656.926,Z 426.303,A 0.000,B 0.000,C 90.000,E1 270.516} C_DIS
LIN {X 0.280,Y -654.340,Z 426.296,A 0.000,B 0.000,C 90.000,E1 269.255} C_DIS
LIN {X -0.049,Y -651.404,Z 426.289,A 0.000,B 0.000,C 90.000,E1 268.051} C_DIS
LIN {X 0.231,Y -648.203,Z 426.282,A 0.000,B 0.000,C 90.000,E1 266.788} C_DIS
LIN {X 0.036,Y -643.490,Z 426.273,A 0.000,B 0.000,C 90.000,E1 265.065} C_DIS
LIN {X -0.232,Y -640.841,Z 426.267,A 0.000,B 0.000,C 90.000,E1 264.090} C_DIS
LIN {X 0.162,Y -638.002,Z 426.262,A 0.000,B 0.000,C 90.000,E1 263.053} C_DIS
LIN {X -0.309,Y -634.171,Z 426.255,A 0.000,B 0.000,C 90.000,E1 261.837} C_DIS
LIN {X 0.207,Y -629.462,Z 426.246,A 0.000,B 0.000,C 90.000,E1 260.274} C_DIS
LIN {X 0.111,Y -624.714,Z 426.238,A 0.000,B 0.000,C 90.000,E1 258.757} C_DIS
LIN {X 0.052,Y -619.827,Z 426.229,A 0.000,B 0.000,C 90.000,E1 257.229} C_DIS
LIN {X -0.239,Y -616.471,Z 426.223,A 0.000,B 0.000,C 90.000,E1 256.228} C_DIS
LIN {X 0.285,Y -611.308,Z 426.215,A 0.000,B 0.000,C 90.000,E1 254.629} C_DIS
LIN {X 0.101,Y -605.849,Z 426.206,A 0.000,B 0.000,C 90.000,E1 253.087} C_DIS
LIN {X 0.253,Y -601.174,Z 426.199,A 0.000,B 0.000,C 90.000,E1 251.764} C_DIS
LIN {X 0.054,Y -597.380,Z 426.193,A 0.000,B 0.000,C 90.000,E1 250.732} C_DIS
LIN {X -0.194,Y -593.451,Z 426.187,A 0.000,B 0.000,C 90.000,E1 249.699} C_DIS
LIN {X 0.151,Y -588.417,Z 426.180,A 0.000,B 0.000,C 90.000,E1 248.337} C_DIS
LIN {X -0.354,Y -583.141,Z 426.172,A 0.000,B 0.000,C 90.000,E1 247.050} C_DIS
LIN {X 0.039,Y -577.758,Z 426.165,A 0.000,B 0.000,C 90.000,E1 245.665} C_DIS
LIN {X -0.183,Y -572.242,Z 426.157,A 0.000,B 0.000,C 90.000,E1 244.332} C_DIS
LIN {X 0.006,Y -566.762,Z 426.150,A 0.000,B 0.000,C 90.000,E1 242.948} C_DIS
LIN {X -0.088,Y -560.130,Z 426.141,A 0.000,B 0.000,C 90.000,E1 241.307} C_DIS
LIN {X -0.090,Y -554.779,Z 426.133,A 0.000,B 0.000,C 90.000,E1 239.921} C_DIS
LIN {X 0.077,Y -547.387,Z 426.122,A 0.000,B 0.000,C 90.000,E1 237.946} C_DIS
LIN {X -0.312,Y -541.266,Z 426.113,A 0.000,B 0.000,C 90.000,E1 236.294} C_DIS
LIN {X -0.072,Y -534.286,Z 426.102,A 0.000,B 0.000,C 90.000,E1 234.276} C_DIS
LIN {X -0.097,Y -529.327,Z 426.094,A 0.000,B 0.000,C 90.000,E1 232.844} C_DIS
LIN {X 0.079,Y -523.345,Z 426.084,A 0.000,B 0.000,C 90.000,E1 231.090} C_DIS
LIN {X 0.041,Y -513.206,Z 426.066,A 0.000,B 0.000,C 90.000,E1 227.877} C_DIS
LIN {X -0.237,Y -508.051,Z 426.056,A 0.000,B 0.000,C 90.000,E1 226.134} C_DIS
LIN {X -0.047,Y -502.107,Z 426.045,A 0.000,B 0.000,C 90.000,E1 224.028} C_DIS
LIN {X 0.003,Y -496.270,Z 426.033,A 0.000,B 0.000,C 90.000,E1 221.919} C_DIS
LIN {X -0.056,Y -490.610,Z 426.021,A 0.000,B 0.000,C 90.000,E1 219.806} C_DIS
LIN {X -0.021,Y -485.932,Z 426.011,A 0.000,B 0.000,C 90.000,E1 217.971} C_DIS
LIN {X 0.101,Y -480.647,Z 425.999,A 0.000,B 0.000,C 90.000,E1 215.804} C_DIS
LIN {X -0.086,Y -475.624,Z 425.987,A 0.000,B 0.000,C 90.000,E1 213.658} C_DIS
LIN {X -0.138,Y -472.849,Z 425.980,A 0.000,B 0.000,C 90.000,E1 212.418} C_DIS
LIN {X 0.013,Y -467.971,Z 425.968,A 0.000,B 0.000,C 90.000,E1 210.207} C_DIS
LIN {X 0.140,Y -464.533,Z 425.959,A 0.000,B 0.000,C 90.000,E1 208.615} C_DIS
LIN {X -0.157,Y -461.713,Z 425.952,A 0.000,B 0.000,C 90.000,E1 207.385} C_DIS
LIN {X -0.067,Y -457.446,Z 425.941,A 0.000,B 0.000,C 90.000,E1 205.463} C_DIS
LIN {X 0.242,Y -453.862,Z 425.933,A 0.000,B 0.000,C 90.000,E1 203.823} C_DIS
LIN {X -0.121,Y -450.229,Z 425.924,A 0.000,B 0.000,C 90.000,E1 202.259} C_DIS
LIN {X -0.017,Y -445.986,Z 425.913,A 0.000,B 0.000,C 90.000,E1 200.301} C_DIS
LIN {X -0.037,Y -440.766,Z 425.898,A 0.000,B 0.000,C 90.000,E1 197.692} C_DIS
LIN {X 0.114,Y -436.677,Z 425.886,A 0.000,B 0.000,C 90.000,E1 195.371} C_DIS
LIN {X 0.165,Y -432.296,Z 425.871,A 0.000,B 0.000,C 90.000,E1 192.715} C_DIS
LIN {X 0.103,Y -429.266,Z 425.860,A 0.000,B 0.000,C 90.000,E1 190.725} C_DIS
LIN {X 0.084,Y -425.629,Z 425.845,A 0.000,B 0.000,C 90.000,E1 188.049} C_DIS
LIN {X -0.181,Y -422.438,Z 425.830,A 0.000,B 0.000,C 90.000,E1 185.391} C_DIS
LIN {X -0.183,Y -419.107,Z 425.811,A 0.000,B 0.000,C 90.000,E1 182.007} C_DIS
LIN {X 0.068,Y -416.935,Z 425.794,A 0.000,B 0.000,C 90.000,E1 178.912} C_DIS
LIN {X -0.079,Y -415.308,Z 425.771,A 0.000,B 0.000,C 90.000,E1 174.837} C_DIS
LIN {X 0.147,Y -415.139,Z 425.758,A 0.000,B 0.000,C 90.000,E1 172.413} C_DIS
LIN {X 0.065,Y -415.593,Z 425.743,A 0.000,B 0.000,C 90.000,E1 169.690} C_DIS
LIN {X -0.143,Y -417.696,Z 425.718,A 0.000,B 0.000,C 90.000,E1 165.283} C_DIS
LIN {X 0.160,Y -420.164,Z 425.701,A 0.000,B 0.000,C 90.000,E1 162.181} C_DIS
LIN {X -0.086,Y -421.506,Z 425.694,A 0.000,B 0.000,C 90.000,E1 160.859} C_DIS
LIN {X 0.096,Y -425.075,Z 425.677,A 0.000,B 0.000,C 90.000,E1 157.794} C_DIS
LIN {X -0.053,Y -429.210,Z 425.660,A 0.000,B 0.000,C 90.000,E1 154.793} C_DIS
LIN {X -0.085,Y -432.425,Z 425.649,A 0.000,B 0.000,C 90.000,E1 152.794} C_DIS
LIN {X 0.038,Y -437.830,Z 425.632,A 0.000,B 0.000,C 90.000,E1 149.793} C_DIS
LIN {X -0.060,Y -442.536,Z 425.619,A 0.000,B 0.000,C 90.000,E1 147.502} C_DIS
LIN {X -0.165,Y -446.144,Z 425.610,A 0.000,B 0.000,C 90.000,E1 145.881} C_DIS
LIN {X 0.127,Y -453.063,Z 425.594,A 0.000,B 0.000,C 90.000,E1 142.924} C_DIS
LIN {X 0.124,Y -459.857,Z 425.580,A 0.000,B 0.000,C 90.000,E1 140.356} C_DIS
LIN {X -0.186,Y -465.138,Z 425.569,A 0.000,B 0.000,C 90.000,E1 138.485} C_DIS
LIN {X -0.180,Y -469.412,Z 425.561,A 0.000,B 0.000,C 90.000,E1 136.905} C_DIS
LIN {X -0.177,Y -472.586,Z 425.554,A 0.000,B 0.000,C 90.000,E1 135.648} C_DIS
LIN {X 0.105,Y -474.826,Z 425.548,A 0.000,B 0.000,C 90.000,E1 134.676} C_DIS
LIN {X -0.154,Y -477.575,Z 425.541,A 0.000,B 0.000,C 90.000,E1 133.461} C_DIS
LIN {X -0.146,Y -479.331,Z 425.536,A 0.000,B 0.000,C 90.000,E1 132.528} C_DIS
LIN {X 0.002,Y -481.266,Z 425.529,A 0.000,B 0.000,C 90.000,E1 131.272} C_DIS
LIN {X 0.099,Y -482.273,Z 425.524,A 0.000,B 0.000,C 90.000,E1 130.334} C_DIS
LIN {X 0.155,Y -482.875,Z 425.519,A 0.000,B 0.000,C 90.000,E1 129.402} C_DIS
LIN {X -0.030,Y -483.011,Z 425.517,A 0.000,B 0.000,C 90.000,E1 129.116} C_DIS
LIN {X 0.100,Y -482.923,Z 425.512,A 0.000,B 0.000,C 90.000,E1 128.177} C_DIS
LIN {X 0.230,Y -482.243,Z 425.507,A 0.000,B 0.000,C 90.000,E1 127.237} C_DIS
LIN {X 0.165,Y -480.652,Z 425.500,A 0.000,B 0.000,C 90.000,E1 126.011} C_DIS
LIN {X 0.177,Y -479.729,Z 425.497,A 0.000,B 0.000,C 90.000,E1 125.391} C_DIS
LIN {X -0.209,Y -478.621,Z 425.493,A 0.000,B 0.000,C 90.000,E1 124.818} C_DIS
LIN {X -0.218,Y -475.597,Z 425.486,A 0.000,B 0.000,C 90.000,E1 123.579} C_DIS
LIN {X -0.239,Y -473.877,Z 425.483,A 0.000,B 0.000,C 90.000,E1 122.959} C_DIS
LIN {X -0.097,Y -470.986,Z 425.478,A 0.000,B 0.000,C 90.000,E1 122.005} C_DIS
LIN {X 0.166,Y -466.729,Z 425.471,A 0.000,B 0.000,C 90.000,E1 120.718} C_DIS
LIN {X -0.022,Y -463.209,Z 425.466,A 0.000,B 0.000,C 90.000,E1 119.795} C_DIS
LIN {X 0.020,Y -457.516,Z 425.458,A 0.000,B 0.000,C 90.000,E1 118.359} C_DIS
LIN {X -0.131,Y -452.938,Z 425.451,A 0.000,B 0.000,C 90.000,E1 117.257} C_DIS
LIN {X 0.258,Y -446.163,Z 425.442,A 0.000,B 0.000,C 90.000,E1 115.591} C_DIS
LIN {X -0.068,Y -444.143,Z 425.440,A 0.000,B 0.000,C 90.000,E1 115.155} C_DIS
LIN {X -0.107,Y -444.144,Z 425.440,A 0.000,B 0.000,C 90.000,E1 115.155} C_DIS
LIN {X 0.173,Y -444.656,Z 425.439,A 0.000,B 0.000,C 90.000,E1 114.951} C_DIS
LIN {X 0.148,Y -454.632,Z 425.415,A 0.000,B 0.000,C 90.000,E1 110.737} C_DIS
LIN {X -0.159,Y -457.292,Z 425.410,A 0.000,B 0.000,C 90.000,E1 109.812} C_DIS
LIN {X -0.091,Y -465.914,Z 425.387,A 0.000,B 0.000,C 90.000,E1 105.662} C_DIS
LIN {X 0.080,Y -467.476,Z 425.383,A 0.000,B 0.000,C 90.000,E1 105.009} C_DIS
LIN {X -0.116,Y -468.077,Z 425.382,A 0.000,B 0.000,C 90.000,E1 104.717} C_DIS
LIN {X 0.024,Y -475.726,Z 425.357,A 0.000,B 0.000,C 90.000,E1 100.310} C_DIS
LIN {X -0.139,Y -476.271,Z 425.356,A 0.000,B 0.000,C 90.000,E1 100.018} C_DIS
LIN {X 0.125,Y -482.156,Z 425.330,A 0.000,B 0.000,C 90.000,E1 95.334} C_DIS
LIN {X -0.120,Y -485.537,Z 425.304,A 0.000,B 0.000,C 90.000,E1 90.745} C_DIS
LIN {X 0.087,Y -486.301,Z 425.282,A 0.000,B 0.000,C 90.000,E1 86.731} C_DIS
LIN {X 0.222,Y -486.330,Z 425.279,A 0.000,B 0.000,C 90.000,E1 86.102} C_DIS
LIN {X -0.185,Y -484.636,Z 425.253,A 0.000,B 0.000,C 90.000,E1 81.546} C_DIS
LIN {X 0.174,Y -480.562,Z 425.227,A 0.000,B 0.000,C 90.000,E1 76.881} C_DIS
LIN {X 0.084,Y -474.320,Z 425.201,A 0.000,B 0.000,C 90.000,E1 72.236} C_DIS
LIN {X -0.095,Y -473.922,Z 425.200,A 0.000,B 0.000,C 90.000,E1 71.945} C_DIS
LIN {X -0.100,Y -466.210,Z 425.175,A 0.000,B 0.000,C 90.000,E1 67.486} C_DIS
LIN {X -0.140,Y -466.231,Z 425.175,A 0.000,B 0.000,C 90.000,E1 67.486} C_DIS
LIN {X -0.013,Y -477.501,Z 425.167,A 0.000,B 0.000,C 90.000,E1 65.973} C_DIS
LIN {X 0.165,Y -483.387,Z 425.162,A 0.000,B 0.000,C 90.000,E1 65.177} C_DIS
LIN {X -0.265,Y -491.341,Z 425.156,A 0.000,B 0.000,C 90.000,E1 64.152} C_DIS
LIN {X 0.009,Y -495.739,Z 425.153,A 0.000,B 0.000,C 90.000,E1 63.512} C_DIS
LIN {X -0.125,Y -499.836,Z 425.150,A 0.000,B 0.000,C 90.000,E1 62.922} C_DIS
LIN {X 0.222,Y -503.668,Z 425.146,A 0.000,B 0.000,C 90.000,E1 62.281} C_DIS
LIN {X -0.089,Y -507.225,Z 425.143,A 0.000,B 0.000,C 90.000,E1 61.719} C_DIS
LIN {X -0.137,Y -510.496,Z 425.140,A 0.000,B 0.000,C 90.000,E1 61.129} C_DIS
LIN {X -0.163,Y -513.544,Z 425.136,A 0.000,B 0.000,C 90.000,E1 60.539} C_DIS
LIN {X 0.094,Y -516.328,Z 425.133,A 0.000,B 0.000,C 90.000,E1 59.921} C_DIS
LIN {X 0.116,Y -518.812,Z 425.130,A 0.000,B 0.000,C 90.000,E1 59.331} C_DIS
LIN {X 0.151,Y -520.929,Z 425.126,A 0.000,B 0.000,C 90.000,E1 58.742} C_DIS
LIN {X 0.139,Y -523.510,Z 425.122,A 0.000,B 0.000,C 90.000,E1 57.867} C_DIS
LIN {X -0.243,Y -524.903,Z 425.118,A 0.000,B 0.000,C 90.000,E1 57.327} C_DIS
LIN {X 0.075,Y -526.490,Z 425.114,A 0.000,B 0.000,C 90.000,E1 56.421} C_DIS
LIN {X 0.117,Y -527.491,Z 425.109,A 0.000,B 0.000,C 90.000,E1 55.548} C_DIS
LIN {X 0.059,Y -528.002,Z 425.105,A 0.000,B 0.000,C 90.000,E1 54.975} C_DIS
LIN {X -0.015,Y -528.271,Z 425.101,A 0.000,B 0.000,C 90.000,E1 54.116} C_DIS
LIN {X -0.082,Y -528.160,Z 425.096,A 0.000,B 0.000,C 90.000,E1 53.256} C_DIS
LIN {X -0.149,Y -527.827,Z 425.091,A 0.000,B 0.000,C 90.000,E1 52.396} C_DIS
LIN {X -0.251,Y -527.048,Z 425.085,A 0.000,B 0.000,C 90.000,E1 51.251} C_DIS
LIN {X -0.039,Y -526.006,Z 425.078,A 0.000,B 0.000,C 90.000,E1 50.070} C_DIS
LIN {X -0.246,Y -524.727,Z 425.072,A 0.000,B 0.000,C 90.000,E1 48.933} C_DIS
LIN {X -0.034,Y -523.668,Z 425.067,A 0.000,B 0.000,C 90.000,E1 48.038} C_DIS
LIN {X -0.010,Y -521.693,Z 425.059,A 0.000,B 0.000,C 90.000,E1 46.581} C_DIS
LIN {X 0.041,Y -518.255,Z 425.044,A 0.000,B 0.000,C 90.000,E1 43.947} C_DIS
LIN {X -0.187,Y -515.884,Z 425.033,A 0.000,B 0.000,C 90.000,E1 41.919} C_DIS
LIN {X -0.097,Y -513.605,Z 425.021,A 0.000,B 0.000,C 90.000,E1 39.850} C_DIS
LIN {X -0.249,Y -511.642,Z 425.012,A 0.000,B 0.000,C 90.000,E1 38.096} C_DIS
LIN {X 0.051,Y -509.925,Z 425.003,A 0.000,B 0.000,C 90.000,E1 36.583} C_DIS
LIN {X -0.080,Y -507.756,Z 424.993,A 0.000,B 0.000,C 90.000,E1 34.818} C_DIS
LIN {X 0.257,Y -505.846,Z 424.985,A 0.000,B 0.000,C 90.000,E1 33.293} C_DIS
LIN {X 0.279,Y -503.866,Z 424.977,A 0.000,B 0.000,C 90.000,E1 31.799} C_DIS
LIN {X 0.003,Y -501.844,Z 424.969,A 0.000,B 0.000,C 90.000,E1 30.335} C_DIS
LIN {X -0.022,Y -499.470,Z 424.959,A 0.000,B 0.000,C 90.000,E1 28.537} C_DIS
LIN {X 0.134,Y -496.866,Z 424.947,A 0.000,B 0.000,C 90.000,E1 26.411} C_DIS
LIN {X -0.157,Y -494.213,Z 424.933,A 0.000,B 0.000,C 90.000,E1 24.027} C_DIS
LIN {X 0.011,Y -491.514,Z 424.917,A 0.000,B 0.000,C 90.000,E1 20.972} C_DIS
LIN {X -0.086,Y -490.036,Z 424.905,A 0.000,B 0.000,C 90.000,E1 18.852} C_DIS
LIN {X -0.134,Y -489.243,Z 424.898,A 0.000,B 0.000,C 90.000,E1 17.638} C_DIS
LIN {X 0.022,Y -487.713,Z 424.886,A 0.000,B 0.000,C 90.000,E1 15.481} C_DIS
LIN {X -0.121,Y -486.330,Z 424.874,A 0.000,B 0.000,C 90.000,E1 13.355} C_DIS
LIN {X 0.191,Y -485.430,Z 424.864,A 0.000,B 0.000,C 90.000,E1 11.478} C_DIS
LIN {X 0.260,Y -484.710,Z 424.852,A 0.000,B 0.000,C 90.000,E1 9.321} C_DIS
LIN {X 0.021,Y -484.275,Z 424.838,A 0.000,B 0.000,C 90.000,E1 6.891} C_DIS
LIN {X 0.144,Y -484.383,Z 424.825,A 0.000,B 0.000,C 90.000,E1 4.416} C_DIS
LIN {X 0.155,Y -486.184,Z 424.801,A 0.000,B 0.000,C 90.000,E1 0.115} C_DIS
LIN {X 0.164,Y -490.172,Z 424.779,A 0.000,B 0.000,C 90.000,E1 356.102} C_DIS
LIN {X -0.101,Y -493.828,Z 424.763,A 0.000,B 0.000,C 90.000,E1 353.394} C_DIS
LIN {X 0.074,Y -497.165,Z 424.751,A 0.000,B 0.000,C 90.000,E1 351.254} C_DIS
LIN {X -0.081,Y -500.823,Z 424.740,A 0.000,B 0.000,C 90.000,E1 349.162} C_DIS
LIN {X -0.112,Y -510.332,Z 424.715,A 0.000,B 0.000,C 90.000,E1 344.685} C_DIS
LIN {X -0.077,Y -514.600,Z 424.705,A 0.000,B 0.000,C 90.000,E1 342.906} C_DIS
LIN {X -0.137,Y -519.135,Z 424.695,A 0.000,B 0.000,C 90.000,E1 341.148} C_DIS
LIN {X -0.249,Y -523.064,Z 424.687,A 0.000,B 0.000,C 90.000,E1 339.699} C_DIS
LIN {X 0.056,Y -527.938,Z 424.677,A 0.000,B 0.000,C 90.000,E1 337.922} C_DIS
LIN {X 0.080,Y -534.427,Z 424.665,A 0.000,B 0.000,C 90.000,E1 335.613} C_DIS
LIN {X 0.084,Y -539.466,Z 424.655,A 0.000,B 0.000,C 90.000,E1 333.896} C_DIS
LIN {X 0.192,Y -545.449,Z 424.644,A 0.000,B 0.000,C 90.000,E1 331.897} C_DIS
LIN {X -0.036,Y -549.846,Z 424.636,A 0.000,B 0.000,C 90.000,E1 330.511} C_DIS
LIN {X 0.057,Y -555.162,Z 424.627,A 0.000,B 0.000,C 90.000,E1 328.820} C_DIS
LIN {X -0.116,Y -560.298,Z 424.618,A 0.000,B 0.000,C 90.000,E1 327.168} C_DIS
LIN {X -0.271,Y -564.536,Z 424.610,A 0.000,B 0.000,C 90.000,E1 325.801} C_DIS
LIN {X -0.035,Y -568.860,Z 424.602,A 0.000,B 0.000,C 90.000,E1 324.402} C_DIS
LIN {X 0.097,Y -574.867,Z 424.592,A 0.000,B 0.000,C 90.000,E1 322.477} C_DIS
LIN {X -0.088,Y -581.078,Z 424.581,A 0.000,B 0.000,C 90.000,E1 320.598} C_DIS
LIN {X -0.011,Y -586.509,Z 424.572,A 0.000,B 0.000,C 90.000,E1 318.976} C_DIS
LIN {X -0.200,Y -591.859,Z 424.563,A 0.000,B 0.000,C 90.000,E1 317.391} C_DIS
LIN {X -0.100,Y -596.388,Z 424.556,A 0.000,B 0.000,C 90.000,E1 316.053} C_DIS
LIN {X 0.074,Y -600.940,Z 424.549,A 0.000,B 0.000,C 90.000,E1 314.717} C_DIS
LIN {X 0.131,Y -606.395,Z 424.540,A 0.000,B 0.000,C 90.000,E1 313.137} C_DIS
LIN {X -0.110,Y -611.792,Z 424.531,A 0.000,B 0.000,C 90.000,E1 311.595} C_DIS
LIN {X -0.077,Y -616.223,Z 424.524,A 0.000,B 0.000,C 90.000,E1 310.297} C_DIS
LIN {X 0.112,Y -620.531,Z 424.517,A 0.000,B 0.000,C 90.000,E1 308.991} C_DIS
LIN {X -0.105,Y -624.677,Z 424.510,A 0.000,B 0.000,C 90.000,E1 307.729} C_DIS
LIN {X -0.117,Y -627.858,Z 424.504,A 0.000,B 0.000,C 90.000,E1 306.710} C_DIS
LIN {X -0.106,Y -632.439,Z 424.495,A 0.000,B 0.000,C 90.000,E1 305.185} C_DIS
LIN {X -0.014,Y -636.102,Z 424.488,A 0.000,B 0.000,C 90.000,E1 303.913} C_DIS
LIN {X -0.183,Y -640.379,Z 424.480,A 0.000,B 0.000,C 90.000,E1 302.418} C_DIS
LIN {X 0.219,Y -643.852,Z 424.473,A 0.000,B 0.000,C 90.000,E1 301.131} C_DIS
LIN {X -0.052,Y -648.402,Z 424.463,A 0.000,B 0.000,C 90.000,E1 299.411} C_DIS
LIN {X 0.050,Y -650.857,Z 424.458,A 0.000,B 0.000,C 90.000,E1 298.409} C_DIS
LIN {X -0.030,Y -653.804,Z 424.451,A 0.000,B 0.000,C 90.000,E1 297.180} C_DIS
LIN {X -0.239,Y -657.116,Z 424.443,A 0.000,B 0.000,C 90.000,E1 295.720} C_DIS
LIN {X 0.093,Y -659.722,Z 424.436,A 0.000,B 0.000,C 90.000,E1 294.463} C_DIS
LIN {X -0.267,Y -661.655,Z 424.431,A 0.000,B 0.000,C 90.000,E1 293.515} C_DIS
LIN {X 0.000,Y -663.527,Z 424.425,A 0.000,B 0.000,C 90.000,E1 292.514} C_DIS
LIN {X 0.176,Y -665.490,Z 424.418,A 0.000,B 0.000,C 90.000,E1 291.280} C_DIS
LIN {X 0.244,Y -667.049,Z 424.413,A 0.000,B 0.000,C 90.000,E1 290.301} C_DIS
LIN {X 0.245,Y -668.533,Z 424.406,A 0.000,B 0.000,C 90.000,E1 289.087} C_DIS
LIN {X 0.265,Y -669.639,Z 424.399,A 0.000,B 0.000,C 90.000,E1 287.873} C_DIS
LIN {X 0.043,Y -670.114,Z 424.395,A 0.000,B 0.000,C 90.000,E1 287.166} C_DIS
LIN {X -0.110,Y -670.634,Z 424.389,A 0.000,B 0.000,C 90.000,E1 285.969} C_DIS
LIN {X -0.197,Y -670.918,Z 424.383,A 0.000,B 0.000,C 90.000,E1 285.009} C_DIS
LIN {X 0.128,Y -671.044,Z 424.377,A 0.000,B 0.000,C 90.000,E1 283.772} C_DIS
LIN {X -0.264,Y -670.823,Z 424.369,A 0.000,B 0.000,C 90.000,E1 282.355} C_DIS
LIN {X -0.014,Y -670.527,Z 424.363,A 0.000,B 0.000,C 90.000,E1 281.366} C_DIS
LIN {X 0.094,Y -669.874,Z 424.355,A 0.000,B 0.000,C 90.000,E1 279.905} C_DIS
LIN {X 0.150,Y -668.976,Z 424.348,A 0.000,B 0.000,C 90.000,E1 278.690} C_DIS
LIN {X 0.105,Y -667.830,Z 424.340,A 0.000,B 0.000,C 90.000,E1 277.239} C_DIS
LIN {X -0.266,Y -667.136,Z 424.336,A 0.000,B 0.000,C 90.000,E1 276.543} C_DIS
LIN {X -0.025,Y -665.159,Z 424.327,A 0.000,B 0.000,C 90.000,E1 274.821} C_DIS
LIN {X -0.127,Y -663.517,Z 424.320,A 0.000,B 0.000,C 90.000,E1 273.612} C_DIS
LIN {X 0.003,Y -660.734,Z 424.311,A 0.000,B 0.000,C 90.000,E1 271.892} C_DIS
LIN {X -0.221,Y -658.483,Z 424.304,A 0.000,B 0.000,C 90.000,E1 270.688} C_DIS
LIN {X -0.119,Y -657.024,Z 424.300,A 0.000,B 0.000,C 90.000,E1 269.943} C_DIS
LIN {X -0.225,Y -654.912,Z 424.294,A 0.000,B 0.000,C 90.000,E1 268.969} C_DIS
LIN {X 0.312,Y -652.646,Z 424.289,A 0.000,B 0.000,C 90.000,E1 267.936} C_DIS
LIN {X -0.039,Y -649.468,Z 424.282,A 0.000,B 0.000,C 90.000,E1 266.731} C_DIS
LIN {X -0.028,Y -645.522,Z 424.274,A 0.000,B 0.000,C 90.000,E1 265.241} C_DIS
LIN {X 0.185,Y -642.202,Z 424.267,A 0.000,B 0.000,C 90.000,E1 263.976} C_DIS
LIN {X -0.042,Y -639.332,Z 424.261,A 0.000,B 0.000,C 90.000,E1 262.996} C_DIS
LIN {X -0.219,Y -636.341,Z 424.256,A 0.000,B 0.000,C 90.000,E1 262.008} C_DIS
LIN {X -0.083,Y -632.441,Z 424.249,A 0.000,B 0.000,C 90.000,E1 260.735} C_DIS
LIN {X -0.112,Y -627.702,Z 424.240,A 0.000,B 0.000,C 90.000,E1 259.218} C_DIS
LIN {X -0.234,Y -622.846,Z 424.232,A 0.000,B 0.000,C 90.000,E1 257.701} C_DIS
LIN {X -0.104,Y -618.718,Z 424.224,A 0.000,B 0.000,C 90.000,E1 256.408} C_DIS
LIN {X 0.105,Y -614.413,Z 424.217,A 0.000,B 0.000,C 90.000,E1 255.102} C_DIS
LIN {X 0.243,Y -609.946,Z 424.210,A 0.000,B 0.000,C 90.000,E1 253.795} C_DIS
LIN {X -0.285,Y -605.347,Z 424.203,A 0.000,B 0.000,C 90.000,E1 252.543} C_DIS
LIN {X -0.137,Y -600.634,Z 424.196,A 0.000,B 0.000,C 90.000,E1 251.221} C_DIS
LIN {X -0.342,Y -596.740,Z 424.190,A 0.000,B 0.000,C 90.000,E1 250.188} C_DIS
LIN {X 0.165,Y -592.767,Z 424.184,A 0.000,B 0.000,C 90.000,E1 249.082} C_DIS
LIN {X 0.067,Y -588.647,Z 424.178,A 0.000,B 0.000,C 90.000,E1 248.028} C_DIS
LIN {X 0.331,Y -583.334,Z 424.171,A 0.000,B 0.000,C 90.000,E1 246.666} C_DIS
LIN {X 0.099,Y -578.995,Z 424.165,A 0.000,B 0.000,C 90.000,E1 245.613} C_DIS
LIN {X -0.264,Y -572.362,Z 424.156,A 0.000,B 0.000,C 90.000,E1 244.024} C_DIS
LIN {X 0.181,Y -566.883,Z 424.148,A 0.000,B 0.000,C 90.000,E1 242.615} C_DIS
LIN {X -0.310,Y -558.106,Z 424.136,A 0.000,B 0.000,C 90.000,E1 240.461} C_DIS
LIN {X 0.179,Y -551.715,Z 424.126,A 0.000,B 0.000,C 90.000,E1 238.742} C_DIS
LIN {X 0.111,Y -543.492,Z 424.114,A 0.000,B 0.000,C 90.000,E1 236.501} C_DIS
LIN {X -0.023,Y -535.506,Z 424.101,A 0.000,B 0.000,C 90.000,E1 234.242} C_DIS
LIN {X -0.346,Y -529.561,Z 424.092,A 0.000,B 0.000,C 90.000,E1 232.557} C_DIS
LIN {X -0.130,Y -524.607,Z 424.084,A 0.000,B 0.000,C 90.000,E1 231.090} C_DIS
LIN {X -0.114,Y -514.447,Z 424.066,A 0.000,B 0.000,C 90.000,E1 227.877} C_DIS
LIN {X -0.011,Y -509.279,Z 424.056,A 0.000,B 0.000,C 90.000,E1 226.095} C_DIS
LIN {X -0.139,Y -503.329,Z 424.045,A 0.000,B 0.000,C 90.000,E1 224.028} C_DIS
LIN {X -0.057,Y -497.483,Z 424.033,A 0.000,B 0.000,C 90.000,E1 221.919} C_DIS
LIN {X -0.084,Y -491.835,Z 424.021,A 0.000,B 0.000,C 90.000,E1 219.806} C_DIS
LIN {X -0.022,Y -487.124,Z 424.011,A 0.000,B 0.000,C 90.000,E1 217.971} C_DIS
LIN {X -0.076,Y -482.598,Z 424.001,A 0.000,B 0.000,C 90.000,E1 216.137} C_DIS
LIN {X -0.220,Y -477.505,Z 423.989,A 0.000,B 0.000,C 90.000,E1 213.992} C_DIS
LIN {X -0.244,Y -474.735,Z 423.982,A 0.000,B 0.000,C 90.000,E1 212.752} C_DIS
LIN {X -0.044,Y -469.808,Z 423.970,A 0.000,B 0.000,C 90.000,E1 210.541} C_DIS
LIN {X 0.272,Y -465.666,Z 423.959,A 0.000,B 0.000,C 90.000,E1 208.615} C_DIS
LIN {X -0.010,Y -462.821,Z 423.952,A 0.000,B 0.000,C 90.000,E1 207.385} C_DIS
LIN {X 0.105,Y -458.529,Z 423.942,A 0.000,B 0.000,C 90.000,E1 205.463} C_DIS
LIN {X -0.167,Y -454.906,Z 423.933,A 0.000,B 0.000,C 90.000,E1 203.898} C_DIS
LIN {X -0.024,Y -450.508,Z 423.922,A 0.000,B 0.000,C 90.000,E1 201.950} C_DIS
LIN {X 0.215,Y -446.969,Z 423.913,A 0.000,B 0.000,C 90.000,E1 200.301} C_DIS
LIN {X 0.221,Y -441.669,Z 423.898,A 0.000,B 0.000,C 90.000,E1 197.692} C_DIS
LIN {X -0.028,Y -437.565,Z 423.886,A 0.000,B 0.000,C 90.000,E1 195.426} C_DIS
LIN {X -0.159,Y -432.657,Z 423.869,A 0.000,B 0.000,C 90.000,E1 192.467} C_DIS
LIN {X 0.116,Y -429.589,Z 423.858,A 0.000,B 0.000,C 90.000,E1 190.433} C_DIS
LIN {X -0.090,Y -426.861,Z 423.847,A 0.000,B 0.000,C 90.000,E1 188.454} C_DIS
LIN {X 0.186,Y -423.227,Z 423.830,A 0.000,B 0.000,C 90.000,E1 185.391} C_DIS
LIN {X -0.160,Y -419.570,Z 423.809,A 0.000,B 0.000,C 90.000,E1 181.718} C_DIS
LIN {X 0.072,Y -417.665,Z 423.794,A 0.000,B 0.000,C 90.000,E1 178.969} C_DIS
LIN {X -0.084,Y -416.083,Z 423.774,A 0.000,B 0.000,C 90.000,E1 175.241} C_DIS
LIN {X 0.208,Y -415.853,Z 423.758,A 0.000,B 0.000,C 90.000,E1 172.470} C_DIS
LIN {X -0.100,Y -416.592,Z 423.738,A 0.000,B 0.000,C 90.000,E1 168.757} C_DIS
LIN {X -0.014,Y -418.397,Z 423.719,A 0.000,B 0.000,C 90.000,E1 165.338} C_DIS
LIN {X 0.136,Y -421.522,Z 423.698,A 0.000,B 0.000,C 90.000,E1 161.583} C_DIS
LIN {X -0.090,Y -425.761,Z 423.677,A 0.000,B 0.000,C 90.000,E1 157.901} C_DIS
LIN {X -0.005,Y -430.417,Z 423.659,A 0.000,B 0.000,C 90.000,E1 154.537} C_DIS
LIN {X -0.196,Y -434.272,Z 423.646,A 0.000,B 0.000,C 90.000,E1 152.231} C_DIS
LIN {X 0.161,Y -439.232,Z 423.631,A 0.000,B 0.000,C 90.000,E1 149.537} C_DIS
LIN {X 0.046,Y -443.321,Z 423.620,A 0.000,B 0.000,C 90.000,E1 147.582} C_DIS
LIN {X -0.047,Y -446.974,Z 423.611,A 0.000,B 0.000,C 90.000,E1 145.960} C_DIS
LIN {X 0.139,Y -451.524,Z 423.600,A 0.000,B 0.000,C 90.000,E1 143.989} C_DIS
LIN {X -0.012,Y -455.626,Z 423.591,A 0.000,B 0.000,C 90.000,E1 142.396} C_DIS
LIN {X -0.056,Y -460.882,Z 423.580,A 0.000,B 0.000,C 90.000,E1 140.481} C_DIS
LIN {X 0.265,Y -465.385,Z 423.572,A 0.000,B 0.000,C 90.000,E1 138.852} C_DIS
LIN {X -0.108,Y -468.891,Z 423.565,A 0.000,B 0.000,C 90.000,E1 137.634} C_DIS
LIN {X -0.115,Y -472.263,Z 423.558,A 0.000,B 0.000,C 90.000,E1 136.377} C_DIS
LIN {X 0.026,Y -476.189,Z 423.549,A 0.000,B 0.000,C 90.000,E1 134.798} C_DIS
LIN {X 0.127,Y -478.965,Z 423.542,A 0.000,B 0.000,C 90.000,E1 133.542} C_DIS
LIN {X -0.050,Y -481.380,Z 423.535,A 0.000,B 0.000,C 90.000,E1 132.324} C_DIS
LIN {X 0.133,Y -483.295,Z 423.528,A 0.000,B 0.000,C 90.000,E1 131.067} C_DIS
LIN {X -0.110,Y -484.222,Z 423.523,A 0.000,B 0.000,C 90.000,E1 130.172} C_DIS
LIN {X -0.034,Y -484.782,Z 423.518,A 0.000,B 0.000,C 90.000,E1 129.241} C_DIS
LIN {X 0.163,Y -484.923,Z 423.516,A 0.000,B 0.000,C 90.000,E1 128.910} C_DIS
LIN {X -0.064,Y -484.752,Z 423.511,A 0.000,B 0.000,C 90.000,E1 128.016} C_DIS
LIN {X 0.085,Y -484.022,Z 423.506,A 0.000,B 0.000,C 90.000,E1 127.076} C_DIS
LIN {X -0.241,Y -482.392,Z 423.499,A 0.000,B 0.000,C 90.000,E1 125.884} C_DIS
LIN {X 0.065,Y -481.404,Z 423.496,A 0.000,B 0.000,C 90.000,E1 125.231} C_DIS
LIN {X 0.084,Y -480.289,Z 423.492,A 0.000,B 0.000,C 90.000,E1 124.612} C_DIS
LIN {X 0.098,Y -477.187,Z 423.486,A 0.000,B 0.000,C 90.000,E1 123.372} C_DIS
LIN {X -0.104,Y -476.374,Z 423.484,A 0.000,B 0.000,C 90.000,E1 123.086} C_DIS
LIN {X 0.064,Y -473.511,Z 423.479,A 0.000,B 0.000,C 90.000,E1 122.133} C_DIS
LIN {X 0.121,Y -469.274,Z 423.472,A 0.000,B 0.000,C 90.000,E1 120.875} C_DIS
LIN {X -0.032,Y -465.771,Z 423.466,A 0.000,B 0.000,C 90.000,E1 119.951} C_DIS
LIN {X 0.156,Y -461.377,Z 423.460,A 0.000,B 0.000,C 90.000,E1 118.821} C_DIS
LIN {X -0.198,Y -456.154,Z 423.453,A 0.000,B 0.000,C 90.000,E1 117.590} C_DIS
LIN {X 0.121,Y -450.047,Z 423.445,A 0.000,B 0.000,C 90.000,E1 116.104} C_DIS
LIN {X 0.073,Y -444.846,Z 423.438,A 0.000,B 0.000,C 90.000,E1 114.899} C_DIS
LIN {X 0.034,Y -444.846,Z 423.438,A 0.000,B 0.000,C 90.000,E1 114.899} C_DIS
LIN {X 0.085,Y -454.166,Z 423.416,A 0.000,B 0.000,C 90.000,E1 110.918} C_DIS
LIN {X 0.202,Y -456.825,Z 423.411,A 0.000,B 0.000,C 90.000,E1 109.939} C_DIS
LIN {X 0.103,Y -457.569,Z 423.409,A 0.000,B 0.000,C 90.000,E1 109.631} C_DIS
LIN {X 0.191,Y -466.269,Z 423.386,A 0.000,B 0.000,C 90.000,E1 105.481} C_DIS
LIN {X -0.208,Y -467.823,Z 423.383,A 0.000,B 0.000,C 90.000,E1 104.898} C_DIS
LIN {X -0.236,Y -476.029,Z 423.357,A 0.000,B 0.000,C 90.000,E1 100.197} C_DIS
LIN {X 0.067,Y -477.355,Z 423.350,A 0.000,B 0.000,C 90.000,E1 98.916} C_DIS
LIN {X 0.037,Y -481.962,Z 423.331,A 0.000,B 0.000,C 90.000,E1 95.511} C_DIS
LIN {X 0.170,Y -482.350,Z 423.327,A 0.000,B 0.000,C 90.000,E1 94.878} C_DIS
LIN {X -0.178,Y -485.421,Z 423.305,A 0.000,B 0.000,C 90.000,E1 90.917} C_DIS
LIN {X -0.040,Y -485.506,Z 423.302,A 0.000,B 0.000,C 90.000,E1 90.286} C_DIS
LIN {X -0.145,Y -486.372,Z 423.281,A 0.000,B 0.000,C 90.000,E1 86.617} C_DIS
LIN {X 0.165,Y -486.367,Z 423.279,A 0.000,B 0.000,C 90.000,E1 86.274} C_DIS
LIN {X -0.006,Y -485.229,Z 423.268,A 0.000,B 0.000,C 90.000,E1 84.147} C_DIS
LIN {X 0.253,Y -484.691,Z 423.254,A 0.000,B 0.000,C 90.000,E1 81.659} C_DIS
LIN {X 0.050,Y -484.469,Z 423.252,A 0.000,B 0.000,C 90.000,E1 81.376} C_DIS
LIN {X 0.055,Y -480.654,Z 423.228,A 0.000,B 0.000,C 90.000,E1 77.061} C_DIS
LIN {X 0.020,Y -480.389,Z 423.227,A 0.000,B 0.000,C 90.000,E1 76.756} C_DIS
LIN {X -0.206,Y -474.179,Z 423.201,A 0.000,B 0.000,C 90.000,E1 72.127} C_DIS
LIN {X -0.048,Y -471.761,Z 423.194,A 0.000,B 0.000,C 90.000,E1 70.859} C_DIS
LIN {X -0.101,Y -466.537,Z 423.176,A 0.000,B 0.000,C 90.000,E1 67.720} C_DIS
LIN {X -0.141,Y -466.536,Z 423.176,A 0.000,B 0.000,C 90.000,E1 67.720} C_DIS
LIN {X 0.119,Y -479.457,Z 423.167,A 0.000,B 0.000,C 90.000,E1 65.973} C_DIS
LIN {X 0.098,Y -486.535,Z 423.161,A 0.000,B 0.000,C 90.000,E1 65.049} C_DIS
LIN {X -0.085,Y -493.279,Z 423.156,A 0.000,B 0.000,C 90.000,E1 64.152} C_DIS
LIN {X 0.205,Y -497.601,Z 423.153,A 0.000,B 0.000,C 90.000,E1 63.512} C_DIS
LIN {X -0.107,Y -502.601,Z 423.149,A 0.000,B 0.000,C 90.000,E1 62.794} C_DIS
LIN {X 0.076,Y -507.241,Z 423.145,A 0.000,B 0.000,C 90.000,E1 62.025} C_DIS
LIN {X -0.151,Y -511.378,Z 423.141,A 0.000,B 0.000,C 90.000,E1 61.307} C_DIS
LIN {X -0.166,Y -514.456,Z 423.137,A 0.000,B 0.000,C 90.000,E1 60.717} C_DIS
LIN {X -0.158,Y -517.249,Z 423.134,A 0.000,B 0.000,C 90.000,E1 60.127} C_DIS
LIN {X -0.132,Y -519.706,Z 423.131,A 0.000,B 0.000,C 90.000,E1 59.537} C_DIS
LIN {X -0.092,Y -521.892,Z 423.127,A 0.000,B 0.000,C 90.000,E1 58.948} C_DIS
LIN {X 0.234,Y -523.723,Z 423.124,A 0.000,B 0.000,C 90.000,E1 58.329} C_DIS
LIN {X -0.095,Y -524.587,Z 423.123,A 0.000,B 0.000,C 90.000,E1 58.074} C_DIS
LIN {X 0.216,Y -526.616,Z 423.118,A 0.000,B 0.000,C 90.000,E1 57.168} C_DIS
LIN {X -0.143,Y -527.698,Z 423.115,A 0.000,B 0.000,C 90.000,E1 56.628} C_DIS
LIN {X -0.086,Y -528.761,Z 423.110,A 0.000,B 0.000,C 90.000,E1 55.754} C_DIS
LIN {X -0.135,Y -529.255,Z 423.107,A 0.000,B 0.000,C 90.000,E1 55.182} C_DIS
LIN {X -0.177,Y -529.481,Z 423.103,A 0.000,B 0.000,C 90.000,E1 54.609} C_DIS
LIN {X 0.196,Y -529.569,Z 423.099,A 0.000,B 0.000,C 90.000,E1 53.703} C_DIS
LIN {X 0.140,Y -529.303,Z 423.094,A 0.000,B 0.000,C 90.000,E1 52.844} C_DIS
LIN {X 0.082,Y -528.853,Z 423.089,A 0.000,B 0.000,C 90.000,E1 51.984} C_DIS
LIN {X 0.013,Y -528.205,Z 423.084,A 0.000,B 0.000,C 90.000,E1 51.126} C_DIS
LIN {X -0.140,Y -527.422,Z 423.079,A 0.000,B 0.000,C 90.000,E1 50.275} C_DIS
LIN {X 0.076,Y -526.139,Z 423.073,A 0.000,B 0.000,C 90.000,E1 49.094} C_DIS
LIN {X -0.089,Y -525.083,Z 423.068,A 0.000,B 0.000,C 90.000,E1 48.243} C_DIS
LIN {X -0.011,Y -523.098,Z 423.060,A 0.000,B 0.000,C 90.000,E1 46.782} C_DIS
LIN {X -0.293,Y -519.582,Z 423.045,A 0.000,B 0.000,C 90.000,E1 44.190} C_DIS
LIN {X -0.208,Y -516.848,Z 423.032,A 0.000,B 0.000,C 90.000,E1 41.838} C_DIS
LIN {X -0.096,Y -514.521,Z 423.021,A 0.000,B 0.000,C 90.000,E1 39.769} C_DIS
LIN {X -0.230,Y -512.549,Z 423.011,A 0.000,B 0.000,C 90.000,E1 38.016} C_DIS
LIN {X 0.083,Y -510.821,Z 423.003,A 0.000,B 0.000,C 90.000,E1 36.503} C_DIS
LIN {X -0.031,Y -508.644,Z 422.993,A 0.000,B 0.000,C 90.000,E1 34.739} C_DIS
LIN {X 0.042,Y -506.719,Z 422.985,A 0.000,B 0.000,C 90.000,E1 33.245} C_DIS
LIN {X 0.039,Y -505.124,Z 422.978,A 0.000,B 0.000,C 90.000,E1 32.054} C_DIS
LIN {X -0.220,Y -503.112,Z 422.970,A 0.000,B 0.000,C 90.000,E1 30.590} C_DIS
LIN {X -0.165,Y -500.332,Z 422.958,A 0.000,B 0.000,C 90.000,E1 28.487} C_DIS
LIN {X 0.023,Y -497.745,Z 422.947,A 0.000,B 0.000,C 90.000,E1 26.360} C_DIS
LIN {X -0.031,Y -495.102,Z 422.933,A 0.000,B 0.000,C 90.000,E1 23.951} C_DIS
LIN {X -0.063,Y -492.648,Z 422.918,A 0.000,B 0.000,C 90.000,E1 21.227} C_DIS
LIN {X 0.039,Y -491.125,Z 422.906,A 0.000,B 0.000,C 90.000,E1 19.087} C_DIS
LIN {X 0.004,Y -490.333,Z 422.899,A 0.000,B 0.000,C 90.000,E1 17.873} C_DIS
LIN {X 0.293,Y -489.243,Z 422.891,A 0.000,B 0.000,C 90.000,E1 16.315} C_DIS
LIN {X -0.165,Y -488.025,Z 422.881,A 0.000,B 0.000,C 90.000,E1 14.537} C_DIS
LIN {X -0.188,Y -486.394,Z 422.864,A 0.000,B 0.000,C 90.000,E1 11.478} C_DIS
LIN {X 0.259,Y -485.575,Z 422.850,A 0.000,B 0.000,C 90.000,E1 8.973} C_DIS
LIN {X -0.012,Y -485.275,Z 422.836,A 0.000,B 0.000,C 90.000,E1 6.549} C_DIS
LIN {X 0.155,Y -485.466,Z 422.823,A 0.000,B 0.000,C 90.000,E1 4.073} C_DIS
LIN {X 0.185,Y -487.511,Z 422.799,A 0.000,B 0.000,C 90.000,E1 359.771} C_DIS
LIN {X 0.215,Y -491.298,Z 422.779,A 0.000,B 0.000,C 90.000,E1 356.102} C_DIS
LIN {X -0.172,Y -495.437,Z 422.762,A 0.000,B 0.000,C 90.000,E1 353.109} C_DIS
LIN {X -0.129,Y -499.853,Z 422.747,A 0.000,B 0.000,C 90.000,E1 350.387} C_DIS
LIN {X -0.252,Y -504.864,Z 422.732,A 0.000,B 0.000,C 90.000,E1 347.701} C_DIS
LIN {X 0.069,Y -512.282,Z 422.713,A 0.000,B 0.000,C 90.000,E1 344.393} C_DIS
LIN {X -0.102,Y -518.104,Z 422.700,A 0.000,B 0.000,C 90.000,E1 342.054} C_DIS
LIN {X -0.100,Y -523.510,Z 422.689,A 0.000,B 0.000,C 90.000,E1 340.007} C_DIS
LIN {X -0.098,Y -529.165,Z 422.678,A 0.000,B 0.000,C 90.000,E1 337.975} C_DIS
LIN {X 0.058,Y -534.008,Z 422.668,A 0.000,B 0.000,C 90.000,E1 336.230} C_DIS
LIN {X -0.173,Y -539.020,Z 422.658,A 0.000,B 0.000,C 90.000,E1 334.537} C_DIS
LIN {X -0.075,Y -544.104,Z 422.649,A 0.000,B 0.000,C 90.000,E1 332.820} C_DIS
LIN {X -0.103,Y -549.354,Z 422.640,A 0.000,B 0.000,C 90.000,E1 331.129} C_DIS
LIN {X 0.257,Y -554.709,Z 422.630,A 0.000,B 0.000,C 90.000,E1 329.410} C_DIS
LIN {X 0.000,Y -559.048,Z 422.622,A 0.000,B 0.000,C 90.000,E1 328.043} C_DIS
LIN {X 0.300,Y -563.368,Z 422.615,A 0.000,B 0.000,C 90.000,E1 326.628} C_DIS
LIN {X -0.032,Y -569.397,Z 422.604,A 0.000,B 0.000,C 90.000,E1 324.736} C_DIS
LIN {X -0.076,Y -576.292,Z 422.592,A 0.000,B 0.000,C 90.000,E1 322.557} C_DIS
LIN {X 0.310,Y -583.415,Z 422.580,A 0.000,B 0.000,C 90.000,E1 320.356} C_DIS
LIN {X 0.061,Y -588.863,Z 422.571,A 0.000,B 0.000,C 90.000,E1 318.771} C_DIS
LIN {X 0.314,Y -594.271,Z 422.562,A 0.000,B 0.000,C 90.000,E1 317.148} C_DIS
LIN {X 0.246,Y -599.734,Z 422.553,A 0.000,B 0.000,C 90.000,E1 315.567} C_DIS
LIN {X 0.056,Y -604.260,Z 422.546,A 0.000,B 0.000,C 90.000,E1 314.271} C_DIS
LIN {X -0.066,Y -608.825,Z 422.539,A 0.000,B 0.000,C 90.000,E1 312.975} C_DIS
LIN {X 0.199,Y -614.274,Z 422.530,A 0.000,B 0.000,C 90.000,E1 311.391} C_DIS
LIN {X 0.284,Y -618.695,Z 422.523,A 0.000,B 0.000,C 90.000,E1 310.092} C_DIS
LIN {X -0.285,Y -622.175,Z 422.517,A 0.000,B 0.000,C 90.000,E1 309.116} C_DIS
LIN {X 0.010,Y -626.306,Z 422.510,A 0.000,B 0.000,C 90.000,E1 307.810} C_DIS
LIN {X 0.023,Y -629.513,Z 422.504,A 0.000,B 0.000,C 90.000,E1 306.790} C_DIS
LIN {X 0.072,Y -634.112,Z 422.496,A 0.000,B 0.000,C 90.000,E1 305.264} C_DIS
LIN {X -0.186,Y -637.080,Z 422.490,A 0.000,B 0.000,C 90.000,E1 304.278} C_DIS
LIN {X 0.019,Y -641.390,Z 422.482,A 0.000,B 0.000,C 90.000,E1 302.752} C_DIS
LIN {X -0.045,Y -645.614,Z 422.474,A 0.000,B 0.000,C 90.000,E1 301.258} C_DIS
LIN {X 0.194,Y -649.527,Z 422.465,A 0.000,B 0.000,C 90.000,E1 299.745} C_DIS
LIN {X 0.317,Y -652.075,Z 422.460,A 0.000,B 0.000,C 90.000,E1 298.743} C_DIS
LIN {X 0.263,Y -655.052,Z 422.453,A 0.000,B 0.000,C 90.000,E1 297.513} C_DIS
LIN {X -0.038,Y -657.879,Z 422.446,A 0.000,B 0.000,C 90.000,E1 296.309} C_DIS
LIN {X -0.131,Y -660.049,Z 422.441,A 0.000,B 0.000,C 90.000,E1 295.335} C_DIS
LIN {X 0.249,Y -662.633,Z 422.434,A 0.000,B 0.000,C 90.000,E1 294.079} C_DIS
LIN {X -0.200,Y -665.013,Z 422.427,A 0.000,B 0.000,C 90.000,E1 292.898} C_DIS
LIN {X 0.112,Y -666.657,Z 422.422,A 0.000,B 0.000,C 90.000,E1 291.897} C_DIS
LIN {X 0.102,Y -668.566,Z 422.415,A 0.000,B 0.000,C 90.000,E1 290.684} C_DIS
LIN {X 0.218,Y -669.850,Z 422.410,A 0.000,B 0.000,C 90.000,E1 289.704} C_DIS
LIN {X -0.230,Y -671.224,Z 422.402,A 0.000,B 0.000,C 90.000,E1 288.290} C_DIS
LIN {X 0.331,Y -671.860,Z 422.396,A 0.000,B 0.000,C 90.000,E1 287.275} C_DIS
LIN {X 0.261,Y -672.180,Z 422.391,A 0.000,B 0.000,C 90.000,E1 286.315} C_DIS
LIN {X -0.050,Y -672.434,Z 422.384,A 0.000,B 0.000,C 90.000,E1 285.134} C_DIS
LIN {X -0.185,Y -672.463,Z 422.377,A 0.000,B 0.000,C 90.000,E1 283.939} C_DIS
LIN {X -0.051,Y -672.106,Z 422.369,A 0.000,B 0.000,C 90.000,E1 282.479} C_DIS
LIN {X 0.289,Y -671.591,Z 422.363,A 0.000,B 0.000,C 90.000,E1 281.243} C_DIS
LIN {X -0.182,Y -670.924,Z 422.356,A 0.000,B 0.000,C 90.000,E1 280.074} C_DIS
LIN {X -0.116,Y -669.983,Z 422.349,A 0.000,B 0.000,C 90.000,E1 278.859} C_DIS
LIN {X -0.147,Y -668.754,Z 422.341,A 0.000,B 0.000,C 90.000,E1 277.409} C_DIS
LIN {X -0.022,Y -667.830,Z 422.336,A 0.000,B 0.000,C 90.000,E1 276.429} C_DIS
LIN {X -0.255,Y -666.188,Z 422.328,A 0.000,B 0.000,C 90.000,E1 274.992} C_DIS
LIN {X 0.321,Y -664.628,Z 422.321,A 0.000,B 0.000,C 90.000,E1 273.726} C_DIS
LIN {X -0.157,Y -663.504,Z 422.317,A 0.000,B 0.000,C 90.000,E1 273.037} C_DIS
LIN {X 0.321,Y -661.654,Z 422.310,A 0.000,B 0.000,C 90.000,E1 271.776} C_DIS
LIN {X -0.092,Y -659.097,Z 422.302,A 0.000,B 0.000,C 90.000,E1 270.344} C_DIS
LIN {X 0.299,Y -656.610,Z 422.295,A 0.000,B 0.000,C 90.000,E1 269.083} C_DIS
LIN {X 0.203,Y -654.439,Z 422.290,A 0.000,B 0.000,C 90.000,E1 268.108} C_DIS
LIN {X -0.151,Y -651.404,Z 422.283,A 0.000,B 0.000,C 90.000,E1 266.906} C_DIS
LIN {X -0.231,Y -646.896,Z 422.273,A 0.000,B 0.000,C 90.000,E1 265.179} C_DIS
LIN {X 0.017,Y -643.560,Z 422.266,A 0.000,B 0.000,C 90.000,E1 263.913} C_DIS
LIN {X 0.198,Y -640.026,Z 422.259,A 0.000,B 0.000,C 90.000,E1 262.648} C_DIS
LIN {X -0.240,Y -636.201,Z 422.252,A 0.000,B 0.000,C 90.000,E1 261.432} C_DIS
LIN {X -0.010,Y -632.277,Z 422.245,A 0.000,B 0.000,C 90.000,E1 260.151} C_DIS
LIN {X 0.158,Y -628.267,Z 422.238,A 0.000,B 0.000,C 90.000,E1 258.870} C_DIS
LIN {X 0.248,Y -624.228,Z 422.231,A 0.000,B 0.000,C 90.000,E1 257.589} C_DIS
LIN {X -0.209,Y -620.094,Z 422.224,A 0.000,B 0.000,C 90.000,E1 256.353} C_DIS
LIN {X 0.251,Y -616.683,Z 422.218,A 0.000,B 0.000,C 90.000,E1 255.283} C_DIS
LIN {X -0.166,Y -612.232,Z 422.211,A 0.000,B 0.000,C 90.000,E1 254.031} C_DIS
LIN {X -0.071,Y -607.625,Z 422.204,A 0.000,B 0.000,C 90.000,E1 252.725} C_DIS
LIN {X 0.115,Y -602.940,Z 422.197,A 0.000,B 0.000,C 90.000,E1 251.402} C_DIS
LIN {X -0.150,Y -598.053,Z 422.189,A 0.000,B 0.000,C 90.000,E1 250.115} C_DIS
LIN {X 0.168,Y -594.064,Z 422.184,A 0.000,B 0.000,C 90.000,E1 249.028} C_DIS
LIN {X 0.084,Y -589.934,Z 422.178,A 0.000,B 0.000,C 90.000,E1 247.975} C_DIS
LIN {X -0.173,Y -584.594,Z 422.170,A 0.000,B 0.000,C 90.000,E1 246.666} C_DIS
LIN {X 0.145,Y -580.239,Z 422.164,A 0.000,B 0.000,C 90.000,E1 245.561} C_DIS
LIN {X 0.052,Y -573.572,Z 422.155,A 0.000,B 0.000,C 90.000,E1 243.948} C_DIS
LIN {X -0.245,Y -568.087,Z 422.148,A 0.000,B 0.000,C 90.000,E1 242.615} C_DIS
LIN {X -0.008,Y -560.387,Z 422.137,A 0.000,B 0.000,C 90.000,E1 240.667} C_DIS
LIN {X 0.048,Y -553.965,Z 422.128,A 0.000,B 0.000,C 90.000,E1 238.997} C_DIS
LIN {X 0.013,Y -546.695,Z 422.117,A 0.000,B 0.000,C 90.000,E1 237.041} C_DIS
LIN {X 0.063,Y -540.657,Z 422.108,A 0.000,B 0.000,C 90.000,E1 235.341} C_DIS
LIN {X 0.154,Y -534.751,Z 422.098,A 0.000,B 0.000,C 90.000,E1 233.623} C_DIS
LIN {X 0.149,Y -530.825,Z 422.092,A 0.000,B 0.000,C 90.000,E1 232.477} C_DIS
LIN {X 0.056,Y -525.870,Z 422.084,A 0.000,B 0.000,C 90.000,E1 231.045} C_DIS
LIN {X 0.064,Y -515.699,Z 422.066,A 0.000,B 0.000,C 90.000,E1 227.838} C_DIS
LIN {X -0.037,Y -511.394,Z 422.058,A 0.000,B 0.000,C 90.000,E1 226.377} C_DIS
LIN {X 0.238,Y -505.399,Z 422.046,A 0.000,B 0.000,C 90.000,E1 224.271} C_DIS
LIN {X 0.003,Y -499.514,Z 422.035,A 0.000,B 0.000,C 90.000,E1 222.204} C_DIS
LIN {X 0.165,Y -494.646,Z 422.024,A 0.000,B 0.000,C 90.000,E1 220.378} C_DIS
LIN {X -0.102,Y -489.880,Z 422.014,A 0.000,B 0.000,C 90.000,E1 218.588} C_DIS
LIN {X -0.004,Y -485.321,Z 422.004,A 0.000,B 0.000,C 90.000,E1 216.744} C_DIS
LIN {X -0.185,Y -480.155,Z 421.992,A 0.000,B 0.000,C 90.000,E1 214.612} C_DIS
LIN {X -0.179,Y -475.929,Z 421.982,A 0.000,B 0.000,C 90.000,E1 212.752} C_DIS
LIN {X -0.122,Y -471.676,Z 421.971,A 0.000,B 0.000,C 90.000,E1 210.875} C_DIS
LIN {X 0.241,Y -467.517,Z 421.961,A 0.000,B 0.000,C 90.000,E1 208.949} C_DIS
LIN {X 0.129,Y -463.975,Z 421.952,A 0.000,B 0.000,C 90.000,E1 207.385} C_DIS
LIN {X 0.269,Y -459.655,Z 421.942,A 0.000,B 0.000,C 90.000,E1 205.463} C_DIS
LIN {X 0.018,Y -455.990,Z 421.933,A 0.000,B 0.000,C 90.000,E1 203.898} C_DIS
LIN {X 0.014,Y -451.568,Z 421.922,A 0.000,B 0.000,C 90.000,E1 201.972} C_DIS
LIN {X 0.022,Y -447.976,Z 421.913,A 0.000,B 0.000,C 90.000,E1 200.355} C_DIS
LIN {X 0.202,Y -443.291,Z 421.901,A 0.000,B 0.000,C 90.000,E1 198.055} C_DIS
LIN {X -0.171,Y -438.511,Z 421.886,A 0.000,B 0.000,C 90.000,E1 195.481} C_DIS
LIN {X 0.056,Y -433.570,Z 421.869,A 0.000,B 0.000,C 90.000,E1 192.479} C_DIS
LIN {X 0.022,Y -430.495,Z 421.858,A 0.000,B 0.000,C 90.000,E1 190.489} C_DIS
LIN {X -0.165,Y -427.731,Z 421.847,A 0.000,B 0.000,C 90.000,E1 188.511} C_DIS
LIN {X 0.059,Y -424.447,Z 421.832,A 0.000,B 0.000,C 90.000,E1 185.796} C_DIS
LIN {X 0.125,Y -421.276,Z 421.815,A 0.000,B 0.000,C 90.000,E1 182.751} C_DIS
LIN {X 0.027,Y -418.886,Z 421.798,A 0.000,B 0.000,C 90.000,E1 179.714} C_DIS
LIN {X -0.093,Y -417.064,Z 421.778,A 0.000,B 0.000,C 90.000,E1 175.988} C_DIS
LIN {X -0.075,Y -416.647,Z 421.755,A 0.000,B 0.000,C 90.000,E1 171.894} C_DIS
LIN {X 0.069,Y -417.427,Z 421.736,A 0.000,B 0.000,C 90.000,E1 168.465} C_DIS
LIN {X 0.029,Y -419.098,Z 421.719,A 0.000,B 0.000,C 90.000,E1 165.408} C_DIS
LIN {X -0.027,Y -421.567,Z 421.702,A 0.000,B 0.000,C 90.000,E1 162.362} C_DIS
LIN {X -0.134,Y -424.756,Z 421.685,A 0.000,B 0.000,C 90.000,E1 159.337} C_DIS
LIN {X -0.067,Y -427.770,Z 421.672,A 0.000,B 0.000,C 90.000,E1 156.975} C_DIS
LIN {X 0.084,Y -433.894,Z 421.650,A 0.000,B 0.000,C 90.000,E1 152.948} C_DIS
LIN {X -0.100,Y -439.989,Z 421.631,A 0.000,B 0.000,C 90.000,E1 149.665} C_DIS
LIN {X -0.142,Y -444.833,Z 421.619,A 0.000,B 0.000,C 90.000,E1 147.375} C_DIS
LIN {X -0.272,Y -447.773,Z 421.611,A 0.000,B 0.000,C 90.000,E1 146.087} C_DIS
LIN {X -0.064,Y -452.421,Z 421.601,A 0.000,B 0.000,C 90.000,E1 144.116} C_DIS
LIN {X -0.270,Y -460.103,Z 421.585,A 0.000,B 0.000,C 90.000,E1 141.251} C_DIS
LIN {X -0.171,Y -466.455,Z 421.572,A 0.000,B 0.000,C 90.000,E1 139.013} C_DIS
LIN {X 0.131,Y -470.059,Z 421.565,A 0.000,B 0.000,C 90.000,E1 137.715} C_DIS
LIN {X 0.237,Y -474.339,Z 421.557,A 0.000,B 0.000,C 90.000,E1 136.134} C_DIS
LIN {X -0.026,Y -477.477,Z 421.550,A 0.000,B 0.000,C 90.000,E1 134.919} C_DIS
LIN {X -0.244,Y -480.347,Z 421.543,A 0.000,B 0.000,C 90.000,E1 133.704} C_DIS
LIN {X -0.078,Y -482.834,Z 421.536,A 0.000,B 0.000,C 90.000,E1 132.447} C_DIS
LIN {X -0.140,Y -483.913,Z 421.532,A 0.000,B 0.000,C 90.000,E1 131.838} C_DIS
LIN {X -0.060,Y -485.303,Z 421.527,A 0.000,B 0.000,C 90.000,E1 130.906} C_DIS
LIN {X 0.089,Y -486.178,Z 421.522,A 0.000,B 0.000,C 90.000,E1 129.967} C_DIS
LIN {X 0.188,Y -486.697,Z 421.517,A 0.000,B 0.000,C 90.000,E1 129.036} C_DIS
LIN {X 0.016,Y -486.814,Z 421.515,A 0.000,B 0.000,C 90.000,E1 128.749} C_DIS
LIN {X 0.190,Y -486.586,Z 421.510,A 0.000,B 0.000,C 90.000,E1 127.810} C_DIS
LIN {X -0.025,Y -485.763,Z 421.505,A 0.000,B 0.000,C 90.000,E1 126.916} C_DIS
LIN {X -0.154,Y -484.563,Z 421.500,A 0.000,B 0.000,C 90.000,E1 126.011} C_DIS
LIN {X -0.290,Y -483.100,Z 421.495,A 0.000,B 0.000,C 90.000,E1 125.105} C_DIS
LIN {X 0.017,Y -481.957,Z 421.491,A 0.000,B 0.000,C 90.000,E1 124.452} C_DIS
LIN {X 0.051,Y -478.771,Z 421.485,A 0.000,B 0.000,C 90.000,E1 123.214} C_DIS
LIN {X -0.206,Y -476.979,Z 421.481,A 0.000,B 0.000,C 90.000,E1 122.625} C_DIS
LIN {X -0.218,Y -475.006,Z 421.478,A 0.000,B 0.000,C 90.000,E1 122.005} C_DIS
LIN {X 0.109,Y -470.706,Z 421.471,A 0.000,B 0.000,C 90.000,E1 120.718} C_DIS
LIN {X -0.034,Y -467.128,Z 421.466,A 0.000,B 0.000,C 90.000,E1 119.795} C_DIS
LIN {X -0.059,Y -462.692,Z 421.459,A 0.000,B 0.000,C 90.000,E1 118.693} C_DIS
LIN {X 0.110,Y -458.718,Z 421.454,A 0.000,B 0.000,C 90.000,E1 117.719} C_DIS
LIN {X 0.066,Y -452.570,Z 421.446,A 0.000,B 0.000,C 90.000,E1 116.283} C_DIS
LIN {X -0.030,Y -445.406,Z 421.437,A 0.000,B 0.000,C 90.000,E1 114.643} C_DIS
LIN {X -0.070,Y -445.408,Z 421.437,A 0.000,B 0.000,C 90.000,E1 114.643} C_DIS
LIN {X -0.051,Y -454.555,Z 421.416,A 0.000,B 0.000,C 90.000,E1 110.791} C_DIS
LIN {X 0.067,Y -457.225,Z 421.410,A 0.000,B 0.000,C 90.000,E1 109.812} C_DIS
LIN {X 0.136,Y -465.846,Z 421.387,A 0.000,B 0.000,C 90.000,E1 105.662} C_DIS
LIN {X -0.144,Y -467.406,Z 421.384,A 0.000,B 0.000,C 90.000,E1 105.064} C_DIS
LIN {X 0.112,Y -468.038,Z 421.382,A 0.000,B 0.000,C 90.000,E1 104.717} C_DIS
LIN {X 0.253,Y -475.668,Z 421.357,A 0.000,B 0.000,C 90.000,E1 100.310} C_DIS
LIN {X 0.090,Y -476.246,Z 421.356,A 0.000,B 0.000,C 90.000,E1 100.018} C_DIS
LIN {X -0.124,Y -482.138,Z 421.330,A 0.000,B 0.000,C 90.000,E1 95.391} C_DIS
LIN {X 0.110,Y -485.532,Z 421.304,A 0.000,B 0.000,C 90.000,E1 90.745} C_DIS
LIN {X 0.143,Y -486.379,Z 421.280,A 0.000,B 0.000,C 90.000,E1 86.445} C_DIS
LIN {X -0.033,Y -486.345,Z 421.279,A 0.000,B 0.000,C 90.000,E1 86.159} C_DIS
LIN {X 0.045,Y -484.659,Z 421.253,A 0.000,B 0.000,C 90.000,E1 81.546} C_DIS
LIN {X -0.065,Y -480.578,Z 421.227,A 0.000,B 0.000,C 90.000,E1 76.937} C_DIS
LIN {X 0.082,Y -479.148,Z 421.222,A 0.000,B 0.000,C 90.000,E1 75.992} C_DIS
LIN {X 0.133,Y -473.980,Z 421.200,A 0.000,B 0.000,C 90.000,E1 71.945} C_DIS
LIN {X 0.105,Y -466.863,Z 421.177,A 0.000,B 0.000,C 90.000,E1 67.922} C_DIS
LIN {X 0.066,Y -466.889,Z 421.177,A 0.000,B 0.000,C 90.000,E1 67.922} C_DIS
LIN {X -0.119,Y -480.192,Z 421.168,A 0.000,B 0.000,C 90.000,E1 66.177} C_DIS
LIN {X 0.065,Y -487.346,Z 421.162,A 0.000,B 0.000,C 90.000,E1 65.229} C_DIS
LIN {X 0.098,Y -491.864,Z 421.159,A 0.000,B 0.000,C 90.000,E1 64.613} C_DIS
LIN {X -0.028,Y -498.378,Z 421.154,A 0.000,B 0.000,C 90.000,E1 63.717} C_DIS
LIN {X 0.109,Y -503.384,Z 421.150,A 0.000,B 0.000,C 90.000,E1 62.948} C_DIS
LIN {X 0.219,Y -506.248,Z 421.147,A 0.000,B 0.000,C 90.000,E1 62.487} C_DIS
LIN {X 0.166,Y -509.784,Z 421.144,A 0.000,B 0.000,C 90.000,E1 61.897} C_DIS
LIN {X -0.037,Y -513.775,Z 421.140,A 0.000,B 0.000,C 90.000,E1 61.179} C_DIS
LIN {X 0.139,Y -516.045,Z 421.137,A 0.000,B 0.000,C 90.000,E1 60.717} C_DIS
LIN {X 0.160,Y -518.778,Z 421.134,A 0.000,B 0.000,C 90.000,E1 60.127} C_DIS
LIN {X 0.033,Y -521.748,Z 421.130,A 0.000,B 0.000,C 90.000,E1 59.410} C_DIS
LIN {X 0.086,Y -523.894,Z 421.127,A 0.000,B 0.000,C 90.000,E1 58.820} C_DIS
LIN {X -0.020,Y -525.599,Z 421.124,A 0.000,B 0.000,C 90.000,E1 58.250} C_DIS
LIN {X 0.024,Y -527.749,Z 421.119,A 0.000,B 0.000,C 90.000,E1 57.375} C_DIS
LIN {X 0.115,Y -528.858,Z 421.116,A 0.000,B 0.000,C 90.000,E1 56.786} C_DIS
LIN {X 0.040,Y -530.026,Z 421.111,A 0.000,B 0.000,C 90.000,E1 55.928} C_DIS
LIN {X 0.119,Y -530.728,Z 421.106,A 0.000,B 0.000,C 90.000,E1 55.055} C_DIS
LIN {X 0.072,Y -530.910,Z 421.101,A 0.000,B 0.000,C 90.000,E1 54.196} C_DIS
LIN {X 0.032,Y -530.818,Z 421.096,A 0.000,B 0.000,C 90.000,E1 53.336} C_DIS
LIN {X -0.023,Y -530.242,Z 421.090,A 0.000,B 0.000,C 90.000,E1 52.190} C_DIS
LIN {X -0.073,Y -529.616,Z 421.085,A 0.000,B 0.000,C 90.000,E1 51.331} C_DIS
LIN {X 0.199,Y -528.849,Z 421.080,A 0.000,B 0.000,C 90.000,E1 50.436} C_DIS
LIN {X 0.033,Y -527.562,Z 421.074,A 0.000,B 0.000,C 90.000,E1 49.299} C_DIS
LIN {X -0.150,Y -526.101,Z 421.068,A 0.000,B 0.000,C 90.000,E1 48.162} C_DIS
LIN {X -0.052,Y -524.079,Z 421.059,A 0.000,B 0.000,C 90.000,E1 46.701} C_DIS
LIN {X 0.141,Y -520.921,Z 421.047,A 0.000,B 0.000,C 90.000,E1 44.352} C_DIS
LIN {X -0.121,Y -518.138,Z 421.034,A 0.000,B 0.000,C 90.000,E1 42.043} C_DIS
LIN {X 0.148,Y -516.090,Z 421.024,A 0.000,B 0.000,C 90.000,E1 40.253} C_DIS
LIN {X -0.023,Y -514.121,Z 421.014,A 0.000,B 0.000,C 90.000,E1 38.508} C_DIS
LIN {X 0.007,Y -512.412,Z 421.006,A 0.000,B 0.000,C 90.000,E1 37.030} C_DIS
LIN {X -0.009,Y -510.965,Z 420.999,A 0.000,B 0.000,C 90.000,E1 35.851} C_DIS
LIN {X -0.323,Y -509.147,Z 420.991,A 0.000,B 0.000,C 90.000,E1 34.405} C_DIS
LIN {X 0.041,Y -507.181,Z 420.983,A 0.000,B 0.000,C 90.000,E1 32.880} C_DIS
LIN {X 0.140,Y -504.791,Z 420.973,A 0.000,B 0.000,C 90.000,E1 31.082} C_DIS
LIN {X 0.113,Y -501.577,Z 420.960,A 0.000,B 0.000,C 90.000,E1 28.693} C_DIS
LIN {X -0.048,Y -498.630,Z 420.946,A 0.000,B 0.000,C 90.000,E1 26.309} C_DIS
LIN {X -0.067,Y -495.975,Z 420.933,A 0.000,B 0.000,C 90.000,E1 23.898} C_DIS
LIN {X 0.075,Y -493.801,Z 420.919,A 0.000,B 0.000,C 90.000,E1 21.461} C_DIS
LIN {X 0.073,Y -492.031,Z 420.906,A 0.000,B 0.000,C 90.000,E1 19.033} C_DIS
LIN {X 0.084,Y -491.006,Z 420.897,A 0.000,B 0.000,C 90.000,E1 17.511} C_DIS
LIN {X -0.223,Y -489.944,Z 420.889,A 0.000,B 0.000,C 90.000,E1 16.024} C_DIS
LIN {X -0.069,Y -488.951,Z 420.880,A 0.000,B 0.000,C 90.000,E1 14.481} C_DIS
LIN {X -0.051,Y -487.343,Z 420.863,A 0.000,B 0.000,C 90.000,E1 11.422} C_DIS
LIN {X -0.177,Y -486.499,Z 420.848,A 0.000,B 0.000,C 90.000,E1 8.681} C_DIS
LIN {X 0.060,Y -486.295,Z 420.835,A 0.000,B 0.000,C 90.000,E1 6.201} C_DIS
LIN {X -0.099,Y -486.746,Z 420.818,A 0.000,B 0.000,C 90.000,E1 3.154} C_DIS
LIN {X 0.023,Y -489.688,Z 420.792,A 0.000,B 0.000,C 90.000,E1 358.568} C_DIS
LIN {X 0.144,Y -492.787,Z 420.777,A 0.000,B 0.000,C 90.000,E1 355.812} C_DIS
LIN {X -0.173,Y -497.051,Z 420.760,A 0.000,B 0.000,C 90.000,E1 352.818} C_DIS
LIN {X 0.003,Y -501.005,Z 420.747,A 0.000,B 0.000,C 90.000,E1 350.387} C_DIS
LIN {X 0.036,Y -504.863,Z 420.735,A 0.000,B 0.000,C 90.000,E1 348.285} C_DIS
LIN {X 0.275,Y -511.356,Z 420.718,A 0.000,B 0.000,C 90.000,E1 345.283} C_DIS
LIN {X -0.125,Y -514.931,Z 420.710,A 0.000,B 0.000,C 90.000,E1 343.850} C_DIS
LIN {X 0.281,Y -520.877,Z 420.697,A 0.000,B 0.000,C 90.000,E1 341.456} C_DIS
LIN {X -0.130,Y -525.478,Z 420.688,A 0.000,B 0.000,C 90.000,E1 339.752} C_DIS
LIN {X 0.238,Y -530.392,Z 420.678,A 0.000,B 0.000,C 90.000,E1 337.975} C_DIS
LIN {X -0.066,Y -535.257,Z 420.668,A 0.000,B 0.000,C 90.000,E1 336.282} C_DIS
LIN {X 0.006,Y -539.444,Z 420.660,A 0.000,B 0.000,C 90.000,E1 334.845} C_DIS
LIN {X -0.131,Y -545.355,Z 420.649,A 0.000,B 0.000,C 90.000,E1 332.871} C_DIS
LIN {X 0.114,Y -549.747,Z 420.641,A 0.000,B 0.000,C 90.000,E1 331.435} C_DIS
LIN {X -0.013,Y -556.023,Z 420.631,A 0.000,B 0.000,C 90.000,E1 329.488} C_DIS
LIN {X 0.303,Y -561.273,Z 420.621,A 0.000,B 0.000,C 90.000,E1 327.788} C_DIS
LIN {X -0.040,Y -566.440,Z 420.612,A 0.000,B 0.000,C 90.000,E1 326.167} C_DIS
LIN {X -0.112,Y -571.647,Z 420.603,A 0.000,B 0.000,C 90.000,E1 324.529} C_DIS
LIN {X -0.253,Y -577.717,Z 420.592,A 0.000,B 0.000,C 90.000,E1 322.637} C_DIS
LIN {X 0.170,Y -584.847,Z 420.580,A 0.000,B 0.000,C 90.000,E1 320.436} C_DIS
LIN {X 0.141,Y -591.281,Z 420.570,A 0.000,B 0.000,C 90.000,E1 318.566} C_DIS
LIN {X 0.211,Y -597.591,Z 420.560,A 0.000,B 0.000,C 90.000,E1 316.701} C_DIS
LIN {X -0.227,Y -603.071,Z 420.551,A 0.000,B 0.000,C 90.000,E1 315.162} C_DIS
LIN {X 0.117,Y -609.460,Z 420.541,A 0.000,B 0.000,C 90.000,E1 313.299} C_DIS
LIN {X -0.061,Y -614.937,Z 420.532,A 0.000,B 0.000,C 90.000,E1 311.757} C_DIS
LIN {X 0.030,Y -619.446,Z 420.525,A 0.000,B 0.000,C 90.000,E1 310.458} C_DIS
LIN {X -0.205,Y -623.817,Z 420.518,A 0.000,B 0.000,C 90.000,E1 309.197} C_DIS
LIN {X -0.025,Y -628.779,Z 420.509,A 0.000,B 0.000,C 90.000,E1 307.649} C_DIS
LIN {X 0.160,Y -631.175,Z 420.505,A 0.000,B 0.000,C 90.000,E1 306.870} C_DIS
LIN {X 0.236,Y -635.028,Z 420.498,A 0.000,B 0.000,C 90.000,E1 305.598} C_DIS
LIN {X -0.012,Y -638.039,Z 420.492,A 0.000,B 0.000,C 90.000,E1 304.612} C_DIS
LIN {X 0.211,Y -642.400,Z 420.484,A 0.000,B 0.000,C 90.000,E1 303.086} C_DIS
LIN {X 0.166,Y -646.664,Z 420.476,A 0.000,B 0.000,C 90.000,E1 301.592} C_DIS
LIN {X 0.253,Y -649.351,Z 420.470,A 0.000,B 0.000,C 90.000,E1 300.590} C_DIS
LIN {X -0.419,Y -652.655,Z 420.463,A 0.000,B 0.000,C 90.000,E1 299.411} C_DIS
LIN {X -0.152,Y -655.686,Z 420.456,A 0.000,B 0.000,C 90.000,E1 298.153} C_DIS
LIN {X 0.313,Y -658.024,Z 420.451,A 0.000,B 0.000,C 90.000,E1 297.129} C_DIS
LIN {X 0.063,Y -660.845,Z 420.444,A 0.000,B 0.000,C 90.000,E1 295.924} C_DIS
LIN {X 0.004,Y -664.018,Z 420.436,A 0.000,B 0.000,C 90.000,E1 294.463} C_DIS
LIN {X -0.157,Y -666.454,Z 420.429,A 0.000,B 0.000,C 90.000,E1 293.259} C_DIS
LIN {X 0.065,Y -668.498,Z 420.422,A 0.000,B 0.000,C 90.000,E1 292.025} C_DIS
LIN {X 0.326,Y -670.344,Z 420.416,A 0.000,B 0.000,C 90.000,E1 290.791} C_DIS
LIN {X -0.323,Y -671.382,Z 420.412,A 0.000,B 0.000,C 90.000,E1 290.120} C_DIS
LIN {X -0.108,Y -672.743,Z 420.404,A 0.000,B 0.000,C 90.000,E1 288.652} C_DIS
LIN {X -0.169,Y -673.420,Z 420.398,A 0.000,B 0.000,C 90.000,E1 287.692} C_DIS
LIN {X -0.158,Y -673.730,Z 420.394,A 0.000,B 0.000,C 90.000,E1 286.968} C_DIS
LIN {X 0.196,Y -673.939,Z 420.388,A 0.000,B 0.000,C 90.000,E1 285.733} C_DIS
LIN {X 0.151,Y -673.925,Z 420.382,A 0.000,B 0.000,C 90.000,E1 284.773} C_DIS
LIN {X -0.017,Y -673.886,Z 420.378,A 0.000,B 0.000,C 90.000,E1 284.064} C_DIS
LIN {X 0.241,Y -673.296,Z 420.369,A 0.000,B 0.000,C 90.000,E1 282.355} C_DIS
LIN {X -0.200,Y -672.633,Z 420.362,A 0.000,B 0.000,C 90.000,E1 281.186} C_DIS
LIN {X 0.078,Y -671.977,Z 420.357,A 0.000,B 0.000,C 90.000,E1 280.197} C_DIS
LIN {X 0.274,Y -670.993,Z 420.350,A 0.000,B 0.000,C 90.000,E1 278.973} C_DIS
LIN {X 0.343,Y -669.903,Z 420.343,A 0.000,B 0.000,C 90.000,E1 277.757} C_DIS
LIN {X 0.218,Y -668.546,Z 420.335,A 0.000,B 0.000,C 90.000,E1 276.315} C_DIS
LIN {X 0.170,Y -667.218,Z 420.328,A 0.000,B 0.000,C 90.000,E1 275.106} C_DIS
LIN {X 0.219,Y -666.068,Z 420.323,A 0.000,B 0.000,C 90.000,E1 274.131} C_DIS
LIN {X 0.257,Y -664.715,Z 420.318,A 0.000,B 0.000,C 90.000,E1 273.154} C_DIS
LIN {X 0.104,Y -662.976,Z 420.311,A 0.000,B 0.000,C 90.000,E1 271.949} C_DIS
LIN {X -0.260,Y -660.568,Z 420.303,A 0.000,B 0.000,C 90.000,E1 270.516} C_DIS
LIN {X -0.318,Y -658.751,Z 420.297,A 0.000,B 0.000,C 90.000,E1 269.542} C_DIS
LIN {X 0.063,Y -656.201,Z 420.291,A 0.000,B 0.000,C 90.000,E1 268.282} C_DIS
LIN {X 0.159,Y -654.483,Z 420.286,A 0.000,B 0.000,C 90.000,E1 267.535} C_DIS
LIN {X -0.166,Y -651.409,Z 420.280,A 0.000,B 0.000,C 90.000,E1 266.331} C_DIS
LIN {X -0.070,Y -647.600,Z 420.271,A 0.000,B 0.000,C 90.000,E1 264.837} C_DIS
LIN {X 0.181,Y -644.201,Z 420.264,A 0.000,B 0.000,C 90.000,E1 263.571} C_DIS
LIN {X -0.019,Y -641.404,Z 420.259,A 0.000,B 0.000,C 90.000,E1 262.591} C_DIS
LIN {X 0.195,Y -637.592,Z 420.252,A 0.000,B 0.000,C 90.000,E1 261.319} C_DIS
LIN {X 0.001,Y -634.503,Z 420.246,A 0.000,B 0.000,C 90.000,E1 260.330} C_DIS
LIN {X 0.008,Y -629.634,Z 420.238,A 0.000,B 0.000,C 90.000,E1 258.814} C_DIS
LIN {X -0.158,Y -626.435,Z 420.232,A 0.000,B 0.000,C 90.000,E1 257.813} C_DIS
LIN {X -0.171,Y -621.460,Z 420.224,A 0.000,B 0.000,C 90.000,E1 256.284} C_DIS
LIN {X -0.218,Y -618.968,Z 420.219,A 0.000,B 0.000,C 90.000,E1 255.519} C_DIS
LIN {X -0.002,Y -614.546,Z 420.212,A 0.000,B 0.000,C 90.000,E1 254.212} C_DIS
LIN {X -0.123,Y -608.969,Z 420.204,A 0.000,B 0.000,C 90.000,E1 252.670} C_DIS
LIN {X -0.220,Y -605.226,Z 420.198,A 0.000,B 0.000,C 90.000,E1 251.638} C_DIS
LIN {X 0.208,Y -601.331,Z 420.192,A 0.000,B 0.000,C 90.000,E1 250.550} C_DIS
LIN {X -0.082,Y -596.392,Z 420.185,A 0.000,B 0.000,C 90.000,E1 249.263} C_DIS
LIN {X 0.098,Y -591.237,Z 420.177,A 0.000,B 0.000,C 90.000,E1 247.922} C_DIS
LIN {X -0.143,Y -585.851,Z 420.170,A 0.000,B 0.000,C 90.000,E1 246.613} C_DIS
LIN {X -0.101,Y -581.484,Z 420.164,A 0.000,B 0.000,C 90.000,E1 245.537} C_DIS
LIN {X 0.113,Y -574.788,Z 420.155,A 0.000,B 0.000,C 90.000,E1 243.896} C_DIS
LIN {X 0.092,Y -569.290,Z 420.148,A 0.000,B 0.000,C 90.000,E1 242.538} C_DIS
LIN {X 0.362,Y -561.607,Z 420.137,A 0.000,B 0.000,C 90.000,E1 240.589} C_DIS
LIN {X 0.160,Y -555.160,Z 420.128,A 0.000,B 0.000,C 90.000,E1 238.948} C_DIS
LIN {X 0.187,Y -546.895,Z 420.115,A 0.000,B 0.000,C 90.000,E1 236.707} C_DIS
LIN {X -0.185,Y -539.904,Z 420.104,A 0.000,B 0.000,C 90.000,E1 234.769} C_DIS
LIN {X -0.103,Y -534.030,Z 420.095,A 0.000,B 0.000,C 90.000,E1 233.050} C_DIS
LIN {X -0.131,Y -529.107,Z 420.087,A 0.000,B 0.000,C 90.000,E1 231.618} C_DIS
LIN {X 0.063,Y -518.707,Z 420.069,A 0.000,B 0.000,C 90.000,E1 228.405} C_DIS
LIN {X -0.095,Y -513.523,Z 420.059,A 0.000,B 0.000,C 90.000,E1 226.662} C_DIS
LIN {X -0.114,Y -507.474,Z 420.048,A 0.000,B 0.000,C 90.000,E1 224.595} C_DIS
LIN {X 0.204,Y -502.399,Z 420.038,A 0.000,B 0.000,C 90.000,E1 222.771} C_DIS
LIN {X 0.061,Y -497.503,Z 420.028,A 0.000,B 0.000,C 90.000,E1 220.987} C_DIS
LIN {X -0.139,Y -492.679,Z 420.018,A 0.000,B 0.000,C 90.000,E1 219.197} C_DIS
LIN {X -0.227,Y -487.316,Z 420.006,A 0.000,B 0.000,C 90.000,E1 217.076} C_DIS
LIN {X -0.151,Y -481.361,Z 419.992,A 0.000,B 0.000,C 90.000,E1 214.612} C_DIS
LIN {X -0.119,Y -477.122,Z 419.982,A 0.000,B 0.000,C 90.000,E1 212.752} C_DIS
LIN {X -0.034,Y -472.852,Z 419.972,A 0.000,B 0.000,C 90.000,E1 210.875} C_DIS
LIN {X -0.055,Y -468.677,Z 419.961,A 0.000,B 0.000,C 90.000,E1 208.999} C_DIS
LIN {X 0.265,Y -465.129,Z 419.952,A 0.000,B 0.000,C 90.000,E1 207.385} C_DIS
LIN {X -0.068,Y -460.055,Z 419.940,A 0.000,B 0.000,C 90.000,E1 205.207} C_DIS
LIN {X 0.108,Y -456.323,Z 419.931,A 0.000,B 0.000,C 90.000,E1 203.590} C_DIS
LIN {X 0.112,Y -451.904,Z 419.920,A 0.000,B 0.000,C 90.000,E1 201.663} C_DIS
LIN {X -0.120,Y -445.590,Z 419.904,A 0.000,B 0.000,C 90.000,E1 198.779} C_DIS
LIN {X 0.128,Y -440.622,Z 419.890,A 0.000,B 0.000,C 90.000,E1 196.134} C_DIS
LIN {X 0.024,Y -437.163,Z 419.879,A 0.000,B 0.000,C 90.000,E1 194.175} C_DIS
LIN {X 0.064,Y -433.932,Z 419.868,A 0.000,B 0.000,C 90.000,E1 192.187} C_DIS
LIN {X 0.156,Y -430.494,Z 419.855,A 0.000,B 0.000,C 90.000,E1 189.849} C_DIS
LIN {X 0.006,Y -427.312,Z 419.842,A 0.000,B 0.000,C 90.000,E1 187.530} C_DIS
LIN {X 0.049,Y -424.903,Z 419.831,A 0.000,B 0.000,C 90.000,E1 185.511} C_DIS
LIN {X 0.098,Y -422.105,Z 419.816,A 0.000,B 0.000,C 90.000,E1 182.808} C_DIS
LIN {X 0.030,Y -419.685,Z 419.799,A 0.000,B 0.000,C 90.000,E1 179.771} C_DIS
LIN {X -0.006,Y -417.761,Z 419.776,A 0.000,B 0.000,C 90.000,E1 175.698} C_DIS
LIN {X 0.002,Y -417.390,Z 419.755,A 0.000,B 0.000,C 90.000,E1 171.951} C_DIS
LIN {X -0.170,Y -418.297,Z 419.735,A 0.000,B 0.000,C 90.000,E1 168.229} C_DIS
LIN {X -0.015,Y -420.270,Z 419.716,A 0.000,B 0.000,C 90.000,E1 164.810} C_DIS
LIN {X -0.028,Y -421.961,Z 419.704,A 0.000,B 0.000,C 90.000,E1 162.779} C_DIS
LIN {X 0.098,Y -424.681,Z 419.689,A 0.000,B 0.000,C 90.000,E1 160.061} C_DIS
LIN {X 0.203,Y -428.028,Z 419.674,A 0.000,B 0.000,C 90.000,E1 157.358} C_DIS
LIN {X -0.229,Y -432.360,Z 419.658,A 0.000,B 0.000,C 90.000,E1 154.409} C_DIS
LIN {X 0.201,Y -435.804,Z 419.647,A 0.000,B 0.000,C 90.000,E1 152.359} C_DIS
LIN {X 0.012,Y -440.754,Z 419.632,A 0.000,B 0.000,C 90.000,E1 149.744} C_DIS
LIN {X 0.046,Y -446.354,Z 419.617,A 0.000,B 0.000,C 90.000,E1 147.120} C_DIS
LIN {X 0.010,Y -452.536,Z 419.603,A 0.000,B 0.000,C 90.000,E1 144.529} C_DIS
LIN {X -0.054,Y -461.992,Z 419.583,A 0.000,B 0.000,C 90.000,E1 141.009} C_DIS
LIN {X 0.107,Y -468.470,Z 419.571,A 0.000,B 0.000,C 90.000,E1 138.771} C_DIS
LIN {X -0.221,Y -472.078,Z 419.564,A 0.000,B 0.000,C 90.000,E1 137.553} C_DIS
LIN {X -0.179,Y -475.578,Z 419.557,A 0.000,B 0.000,C 90.000,E1 136.296} C_DIS
LIN {X 0.250,Y -478.747,Z 419.550,A 0.000,B 0.000,C 90.000,E1 135.000} C_DIS
LIN {X -0.071,Y -480.987,Z 419.545,A 0.000,B 0.000,C 90.000,E1 134.109} C_DIS
LIN {X 0.110,Y -483.667,Z 419.538,A 0.000,B 0.000,C 90.000,E1 132.852} C_DIS
LIN {X 0.192,Y -485.438,Z 419.533,A 0.000,B 0.000,C 90.000,E1 131.919} C_DIS
LIN {X 0.116,Y -487.266,Z 419.526,A 0.000,B 0.000,C 90.000,E1 130.701} C_DIS
LIN {X -0.082,Y -488.094,Z 419.521,A 0.000,B 0.000,C 90.000,E1 129.806} C_DIS
LIN {X -0.106,Y -488.476,Z 419.518,A 0.000,B 0.000,C 90.000,E1 129.197} C_DIS
LIN {X -0.131,Y -488.665,Z 419.514,A 0.000,B 0.000,C 90.000,E1 128.588} C_DIS
LIN {X 0.063,Y -488.375,Z 419.509,A 0.000,B 0.000,C 90.000,E1 127.649} C_DIS
LIN {X -0.037,Y -487.503,Z 419.504,A 0.000,B 0.000,C 90.000,E1 126.744} C_DIS
LIN {X 0.146,Y -486.284,Z 419.499,A 0.000,B 0.000,C 90.000,E1 125.804} C_DIS
LIN {X -0.195,Y -485.350,Z 419.496,A 0.000,B 0.000,C 90.000,E1 125.231} C_DIS
LIN {X 0.077,Y -483.559,Z 419.491,A 0.000,B 0.000,C 90.000,E1 124.278} C_DIS
LIN {X 0.144,Y -480.352,Z 419.484,A 0.000,B 0.000,C 90.000,E1 123.038} C_DIS
LIN {X 0.158,Y -478.514,Z 419.480,A 0.000,B 0.000,C 90.000,E1 122.418} C_DIS
LIN {X 0.156,Y -476.480,Z 419.477,A 0.000,B 0.000,C 90.000,E1 121.799} C_DIS
LIN {X 0.078,Y -473.284,Z 419.472,A 0.000,B 0.000,C 90.000,E1 120.875} C_DIS
LIN {X 0.138,Y -468.488,Z 419.465,A 0.000,B 0.000,C 90.000,E1 119.617} C_DIS
LIN {X 0.115,Y -463.334,Z 419.458,A 0.000,B 0.000,C 90.000,E1 118.359} C_DIS
LIN {X 0.037,Y -458.612,Z 419.452,A 0.000,B 0.000,C 90.000,E1 117.257} C_DIS
LIN {X -0.213,Y -452.336,Z 419.444,A 0.000,B 0.000,C 90.000,E1 115.848} C_DIS
LIN {X -0.049,Y -445.940,Z 419.435,A 0.000,B 0.000,C 90.000,E1 114.387} C_DIS
LIN {X -0.089,Y -445.947,Z 419.435,A 0.000,B 0.000,C 90.000,E1 114.387} C_DIS
LIN {X 0.239,Y -454.946,Z 419.415,A 0.000,B 0.000,C 90.000,E1 110.610} C_DIS
LIN {X 0.034,Y -456.732,Z 419.411,A 0.000,B 0.000,C 90.000,E1 109.993} C_DIS
LIN {X -0.066,Y -457.510,Z 419.409,A 0.000,B 0.000,C 90.000,E1 109.685} C_DIS
LIN {X -0.121,Y -466.190,Z 419.386,A 0.000,B 0.000,C 90.000,E1 105.552} C_DIS
LIN {X 0.056,Y -467.756,Z 419.383,A 0.000,B 0.000,C 90.000,E1 104.898} C_DIS
LIN {X 0.028,Y -475.962,Z 419.357,A 0.000,B 0.000,C 90.000,E1 100.197} C_DIS
LIN {X 0.177,Y -476.677,Z 419.353,A 0.000,B 0.000,C 90.000,E1 99.557} C_DIS
LIN {X -0.177,Y -481.911,Z 419.331,A 0.000,B 0.000,C 90.000,E1 95.568} C_DIS
LIN {X 0.150,Y -482.202,Z 419.329,A 0.000,B 0.000,C 90.000,E1 95.220} C_DIS
LIN {X 0.088,Y -485.389,Z 419.305,A 0.000,B 0.000,C 90.000,E1 90.917} C_DIS
LIN {X -0.088,Y -485.529,Z 419.303,A 0.000,B 0.000,C 90.000,E1 90.630} C_DIS
LIN {X 0.121,Y -486.357,Z 419.281,A 0.000,B 0.000,C 90.000,E1 86.617} C_DIS
LIN {X -0.055,Y -486.369,Z 419.280,A 0.000,B 0.000,C 90.000,E1 86.331} C_DIS
LIN {X -0.065,Y -485.859,Z 419.275,A 0.000,B 0.000,C 90.000,E1 85.412} C_DIS
LIN {X -0.031,Y -484.692,Z 419.254,A 0.000,B 0.000,C 90.000,E1 81.724} C_DIS
LIN {X -0.163,Y -484.508,Z 419.252,A 0.000,B 0.000,C 90.000,E1 81.432} C_DIS
LIN {X 0.175,Y -480.441,Z 419.227,A 0.000,B 0.000,C 90.000,E1 76.769} C_DIS
LIN {X 0.057,Y -474.209,Z 419.201,A 0.000,B 0.000,C 90.000,E1 72.127} C_DIS
LIN {X -0.010,Y -473.052,Z 419.197,A 0.000,B 0.000,C 90.000,E1 71.511} C_DIS
LIN {X 0.055,Y -467.198,Z 419.179,A 0.000,B 0.000,C 90.000,E1 68.156} C_DIS
LIN {X 0.015,Y -467.208,Z 419.179,A 0.000,B 0.000,C 90.000,E1 68.156} C_DIS
LIN {X 0.140,Y -482.053,Z 419.168,A 0.000,B 0.000,C 90.000,E1 66.177} C_DIS
LIN {X -0.094,Y -489.181,Z 419.163,A 0.000,B 0.000,C 90.000,E1 65.281} C_DIS
LIN {X -0.253,Y -494.745,Z 419.158,A 0.000,B 0.000,C 90.000,E1 64.537} C_DIS
LIN {X -0.152,Y -500.077,Z 419.154,A 0.000,B 0.000,C 90.000,E1 63.768} C_DIS
LIN {X -0.184,Y -506.007,Z 419.149,A 0.000,B 0.000,C 90.000,E1 62.871} C_DIS
LIN {X 0.027,Y -510.550,Z 419.145,A 0.000,B 0.000,C 90.000,E1 62.103} C_DIS
LIN {X -0.100,Y -515.308,Z 419.140,A 0.000,B 0.000,C 90.000,E1 61.229} C_DIS
LIN {X -0.166,Y -517.532,Z 419.138,A 0.000,B 0.000,C 90.000,E1 60.795} C_DIS
LIN {X -0.138,Y -520.206,Z 419.134,A 0.000,B 0.000,C 90.000,E1 60.205} C_DIS
LIN {X -0.093,Y -522.602,Z 419.131,A 0.000,B 0.000,C 90.000,E1 59.616} C_DIS
LIN {X 0.238,Y -524.761,Z 419.128,A 0.000,B 0.000,C 90.000,E1 58.997} C_DIS
LIN {X -0.134,Y -526.539,Z 419.125,A 0.000,B 0.000,C 90.000,E1 58.456} C_DIS
LIN {X -0.047,Y -528.064,Z 419.122,A 0.000,B 0.000,C 90.000,E1 57.867} C_DIS
LIN {X -0.081,Y -528.790,Z 419.120,A 0.000,B 0.000,C 90.000,E1 57.582} C_DIS
LIN {X -0.007,Y -530.435,Z 419.115,A 0.000,B 0.000,C 90.000,E1 56.707} C_DIS
LIN {X -0.063,Y -531.478,Z 419.110,A 0.000,B 0.000,C 90.000,E1 55.849} C_DIS
LIN {X 0.047,Y -531.972,Z 419.107,A 0.000,B 0.000,C 90.000,E1 55.261} C_DIS
LIN {X 0.014,Y -532.209,Z 419.102,A 0.000,B 0.000,C 90.000,E1 54.402} C_DIS
LIN {X -0.012,Y -532.190,Z 419.098,A 0.000,B 0.000,C 90.000,E1 53.543} C_DIS
LIN {X -0.036,Y -531.826,Z 419.093,A 0.000,B 0.000,C 90.000,E1 52.683} C_DIS
LIN {X -0.077,Y -531.034,Z 419.086,A 0.000,B 0.000,C 90.000,E1 51.537} C_DIS
LIN {X 0.195,Y -529.961,Z 419.080,A 0.000,B 0.000,C 90.000,E1 50.356} C_DIS
LIN {X -0.273,Y -529.005,Z 419.075,A 0.000,B 0.000,C 90.000,E1 49.542} C_DIS
LIN {X -0.086,Y -527.519,Z 419.069,A 0.000,B 0.000,C 90.000,E1 48.366} C_DIS
LIN {X 0.044,Y -525.515,Z 419.061,A 0.000,B 0.000,C 90.000,E1 46.905} C_DIS
LIN {X -0.080,Y -522.280,Z 419.048,A 0.000,B 0.000,C 90.000,E1 44.595} C_DIS
LIN {X -0.016,Y -519.099,Z 419.033,A 0.000,B 0.000,C 90.000,E1 41.962} C_DIS
LIN {X 0.004,Y -517.349,Z 419.025,A 0.000,B 0.000,C 90.000,E1 40.496} C_DIS
LIN {X -0.062,Y -515.675,Z 419.017,A 0.000,B 0.000,C 90.000,E1 39.036} C_DIS
LIN {X -0.024,Y -514.366,Z 419.010,A 0.000,B 0.000,C 90.000,E1 37.855} C_DIS
LIN {X 0.014,Y -512.627,Z 419.002,A 0.000,B 0.000,C 90.000,E1 36.377} C_DIS
LIN {X -0.056,Y -510.405,Z 418.992,A 0.000,B 0.000,C 90.000,E1 34.612} C_DIS
LIN {X 0.054,Y -508.458,Z 418.984,A 0.000,B 0.000,C 90.000,E1 33.118} C_DIS
LIN {X -0.088,Y -505.653,Z 418.973,A 0.000,B 0.000,C 90.000,E1 31.052} C_DIS
LIN {X -0.105,Y -502.456,Z 418.959,A 0.000,B 0.000,C 90.000,E1 28.665} C_DIS
LIN {X 0.190,Y -499.528,Z 418.946,A 0.000,B 0.000,C 90.000,E1 26.232} C_DIS
LIN {X 0.187,Y -496.860,Z 418.933,A 0.000,B 0.000,C 90.000,E1 23.823} C_DIS
LIN {X 0.112,Y -494.974,Z 418.921,A 0.000,B 0.000,C 90.000,E1 21.716} C_DIS
LIN {X -0.235,Y -493.517,Z 418.911,A 0.000,B 0.000,C 90.000,E1 19.939} C_DIS
LIN {X -0.194,Y -492.523,Z 418.902,A 0.000,B 0.000,C 90.000,E1 18.417} C_DIS
LIN {X 0.027,Y -491.316,Z 418.892,A 0.000,B 0.000,C 90.000,E1 16.567} C_DIS
LIN {X 0.225,Y -490.084,Z 418.882,A 0.000,B 0.000,C 90.000,E1 14.717} C_DIS
LIN {X -0.079,Y -488.549,Z 418.867,A 0.000,B 0.000,C 90.000,E1 12.007} C_DIS
LIN {X -0.039,Y -487.664,Z 418.853,A 0.000,B 0.000,C 90.000,E1 9.557} C_DIS
LIN {X 0.178,Y -487.327,Z 418.838,A 0.000,B 0.000,C 90.000,E1 6.777} C_DIS
LIN {X -0.083,Y -487.685,Z 418.819,A 0.000,B 0.000,C 90.000,E1 3.440} C_DIS
LIN {X 0.199,Y -490.525,Z 418.794,A 0.000,B 0.000,C 90.000,E1 358.854} C_DIS
LIN {X 0.198,Y -493.926,Z 418.777,A 0.000,B 0.000,C 90.000,E1 355.812} C_DIS
LIN {X -0.076,Y -498.223,Z 418.760,A 0.000,B 0.000,C 90.000,E1 352.818} C_DIS
LIN {X 0.138,Y -502.184,Z 418.747,A 0.000,B 0.000,C 90.000,E1 350.387} C_DIS
LIN {X 0.202,Y -506.112,Z 418.735,A 0.000,B 0.000,C 90.000,E1 348.285} C_DIS
LIN {X -0.040,Y -513.349,Z 418.717,A 0.000,B 0.000,C 90.000,E1 345.046} C_DIS
LIN {X 0.062,Y -517.644,Z 418.707,A 0.000,B 0.000,C 90.000,E1 343.268} C_DIS
LIN {X 0.050,Y -522.925,Z 418.696,A 0.000,B 0.000,C 90.000,E1 341.221} C_DIS
LIN {X -0.101,Y -530.872,Z 418.680,A 0.000,B 0.000,C 90.000,E1 338.337} C_DIS
LIN {X -0.114,Y -535.733,Z 418.670,A 0.000,B 0.000,C 90.000,E1 336.613} C_DIS
LIN {X -0.083,Y -540.744,Z 418.661,A 0.000,B 0.000,C 90.000,E1 334.897} C_DIS
LIN {X 0.058,Y -547.525,Z 418.648,A 0.000,B 0.000,C 90.000,E1 332.615} C_DIS
LIN {X 0.112,Y -552.831,Z 418.639,A 0.000,B 0.000,C 90.000,E1 330.923} C_DIS
LIN {X 0.075,Y -558.237,Z 418.629,A 0.000,B 0.000,C 90.000,E1 329.253} C_DIS
LIN {X 0.157,Y -563.526,Z 418.620,A 0.000,B 0.000,C 90.000,E1 327.582} C_DIS
LIN {X -0.142,Y -568.713,Z 418.611,A 0.000,B 0.000,C 90.000,E1 325.960} C_DIS
LIN {X -0.164,Y -573.915,Z 418.602,A 0.000,B 0.000,C 90.000,E1 324.322} C_DIS
LIN {X -0.064,Y -579.189,Z 418.593,A 0.000,B 0.000,C 90.000,E1 322.683} C_DIS
LIN {X -0.222,Y -587.273,Z 418.579,A 0.000,B 0.000,C 90.000,E1 320.275} C_DIS
LIN {X 0.049,Y -592.819,Z 418.570,A 0.000,B 0.000,C 90.000,E1 318.647} C_DIS
LIN {X 0.155,Y -599.146,Z 418.560,A 0.000,B 0.000,C 90.000,E1 316.782} C_DIS
LIN {X -0.253,Y -604.616,Z 418.551,A 0.000,B 0.000,C 90.000,E1 315.243} C_DIS
LIN {X 0.312,Y -610.128,Z 418.543,A 0.000,B 0.000,C 90.000,E1 313.623} C_DIS
LIN {X 0.152,Y -615.590,Z 418.534,A 0.000,B 0.000,C 90.000,E1 312.081} C_DIS
LIN {X -0.046,Y -619.285,Z 418.528,A 0.000,B 0.000,C 90.000,E1 311.067} C_DIS
LIN {X 0.115,Y -623.711,Z 418.521,A 0.000,B 0.000,C 90.000,E1 309.769} C_DIS
LIN {X 0.237,Y -626.288,Z 418.517,A 0.000,B 0.000,C 90.000,E1 308.991} C_DIS
LIN {X -0.026,Y -631.270,Z 418.508,A 0.000,B 0.000,C 90.000,E1 307.488} C_DIS
LIN {X 0.046,Y -635.965,Z 418.500,A 0.000,B 0.000,C 90.000,E1 305.964} C_DIS
LIN {X 0.207,Y -639.750,Z 418.493,A 0.000,B 0.000,C 90.000,E1 304.692} C_DIS
LIN {X -0.068,Y -644.130,Z 418.485,A 0.000,B 0.000,C 90.000,E1 303.214} C_DIS
LIN {X -0.084,Y -648.413,Z 418.476,A 0.000,B 0.000,C 90.000,E1 301.720} C_DIS
LIN {X 0.023,Y -651.128,Z 418.471,A 0.000,B 0.000,C 90.000,E1 300.718} C_DIS
LIN {X -0.055,Y -654.465,Z 418.464,A 0.000,B 0.000,C 90.000,E1 299.489} C_DIS
LIN {X -0.211,Y -658.101,Z 418.456,A 0.000,B 0.000,C 90.000,E1 298.025} C_DIS
LIN {X -0.171,Y -660.996,Z 418.449,A 0.000,B 0.000,C 90.000,E1 296.796} C_DIS
LIN {X 0.077,Y -663.220,Z 418.443,A 0.000,B 0.000,C 90.000,E1 295.796} C_DIS
LIN {X -0.086,Y -665.888,Z 418.437,A 0.000,B 0.000,C 90.000,E1 294.591} C_DIS
LIN {X -0.215,Y -668.258,Z 418.430,A 0.000,B 0.000,C 90.000,E1 293.387} C_DIS
LIN {X 0.140,Y -669.924,Z 418.424,A 0.000,B 0.000,C 90.000,E1 292.386} C_DIS
